C03651=1225.024,372.969,-76.050,-175.825,7.597,148.237
C03652=1225.028,372.721,-76.016,-175.826,7.594,148.237
C03653=1225.032,372.473,-75.983,-175.827,7.591,148.236
C03654=1225.036,372.225,-75.950,-175.829,7.588,148.236
C03655=1225.040,371.977,-75.917,-175.830,7.586,148.236
C03656=1225.044,371.730,-75.883,-175.831,7.583,148.235
C03657=1225.048,371.482,-75.850,-175.833,7.580,148.235
C03658=1225.052,371.234,-75.817,-175.834,7.577,148.235
C03659=1225.056,370.986,-75.784,-175.835,7.575,148.234
C03660=1225.061,370.739,-75.751,-175.837,7.572,148.234
C03661=1225.065,370.491,-75.718,-175.838,7.569,148.234
C03662=1225.069,370.243,-75.684,-175.839,7.566,148.233
C03663=1225.073,369.995,-75.651,-175.841,7.564,148.233
C03664=1225.077,369.748,-75.618,-175.842,7.561,148.233
C03665=1225.081,369.500,-75.585,-175.843,7.558,148.232
C03666=1225.085,369.252,-75.552,-175.844,7.555,148.232
C03667=1225.090,369.005,-75.519,-175.846,7.553,148.232
C03668=1225.094,368.756,-75.486,-175.847,7.550,148.231
C03669=1225.097,368.509,-75.454,-175.848,7.547,148.231
C03670=1225.101,368.261,-75.421,-175.850,7.544,148.231
C03671=1225.106,368.013,-75.387,-175.851,7.542,148.230
C03672=1225.110,367.766,-75.354,-175.852,7.539,148.230
C03673=1225.114,367.486,-75.317,-175.854,7.535,148.230
C03674=1225.120,367.207,-75.280,-175.856,7.533,148.229
C03675=1225.124,366.927,-75.243,-175.857,7.529,148.229
C03676=1225.129,366.647,-75.205,-175.859,7.527,148.229
C03677=1225.134,366.399,-75.173,-175.860,7.524,148.228
C03678=1225.137,366.152,-75.140,-175.861,7.521,148.228
C03679=1225.141,365.904,-75.107,-175.863,7.519,148.228
C03680=1225.145,365.656,-75.074,-175.864,7.516,148.227
C03681=1225.150,365.408,-75.041,-175.866,7.512,148.227
C03682=1225.154,365.160,-75.008,-175.868,7.510,148.227
C03683=1225.158,364.912,-74.975,-175.869,7.507,148.227
C03684=1225.161,364.665,-74.943,-175.870,7.504,148.226
C03685=1225.166,364.417,-74.910,-175.872,7.502,148.226
C03686=1225.170,364.169,-74.877,-175.873,7.499,148.226
C03687=1225.174,363.921,-74.844,-175.875,7.496,148.225
C03688=1225.178,363.673,-74.811,-175.876,7.494,148.225
C03689=1225.183,363.425,-74.778,-175.878,7.490,148.225
C03690=1225.186,363.178,-74.746,-175.880,7.488,148.225
C03691=1225.191,362.931,-74.713,-175.881,7.485,148.224
C03692=1225.195,362.682,-74.680,-175.883,7.482,148.224
C03693=1225.199,362.435,-74.647,-175.884,7.479,148.224
C03694=1225.203,362.186,-74.615,-175.885,7.477,148.223
C03695=1225.207,361.939,-74.582,-175.887,7.474,148.223
C03696=1225.211,361.691,-74.549,-175.889,7.471,148.223
C03697=1225.216,361.443,-74.517,-175.890,7.468,148.223
C03698=1225.219,361.195,-74.484,-175.892,7.465,148.222
C03699=1225.224,360.947,-74.452,-175.893,7.463,148.222
C03700=1225.228,360.700,-74.419,-175.895,7.460,148.222
C03701=1225.232,360.452,-74.386,-175.896,7.458,148.221
C03702=1225.236,360.204,-74.354,-175.898,7.454,148.221
C03703=1225.240,359.956,-74.321,-175.900,7.452,148.221
C03704=1225.245,359.708,-74.288,-175.901,7.449,148.221
C03705=1225.249,359.460,-74.255,-175.903,7.446,148.220
C03706=1225.253,359.212,-74.223,-175.904,7.444,148.220
C03707=1225.257,358.965,-74.190,-175.906,7.440,148.220
C03708=1225.262,358.717,-74.158,-175.908,7.438,148.220
C03709=1225.265,358.469,-74.125,-175.909,7.435,148.219
C03710=1225.270,358.221,-74.093,-175.910,7.432,148.219
C03711=1225.274,357.973,-74.060,-175.912,7.430,148.219
C03712=1225.277,357.725,-74.028,-175.914,7.426,148.219
C03713=1225.282,357.478,-73.995,-175.916,7.424,148.218
C03714=1225.287,357.230,-73.963,-175.917,7.421,148.218
C03715=1225.290,356.982,-73.931,-175.919,7.418,148.218
C03716=1225.295,356.734,-73.898,-175.920,7.416,148.218
C03717=1225.298,356.486,-73.866,-175.922,7.413,148.217
C03718=1225.302,356.238,-73.833,-175.924,7.410,148.217
C03719=1225.307,355.991,-73.801,-175.925,7.407,148.217
C03720=1225.311,355.743,-73.769,-175.927,7.405,148.217
C03721=1225.315,355.495,-73.736,-175.929,7.401,148.216
C03722=1225.320,355.247,-73.703,-175.931,7.399,148.216
C03723=1225.323,354.999,-73.671,-175.932,7.396,148.216
C03724=1225.328,354.752,-73.639,-175.933,7.393,148.216
C03725=1225.332,354.504,-73.607,-175.936,7.390,148.215
C03726=1225.336,354.255,-73.574,-175.937,7.388,148.215
C03727=1225.340,354.008,-73.542,-175.939,7.385,148.215
C03728=1225.344,353.759,-73.509,-175.941,7.382,148.215
C03729=1225.349,353.512,-73.477,-175.942,7.380,148.215
C03730=1225.353,353.264,-73.445,-175.944,7.377,148.214
C03731=1225.357,353.016,-73.412,-175.946,7.374,148.214
C03732=1225.361,352.768,-73.380,-175.947,7.371,148.214
C03733=1225.366,352.520,-73.348,-175.949,7.369,148.214
C03734=1225.369,352.273,-73.316,-175.951,7.365,148.213
C03735=1225.374,352.025,-73.283,-175.953,7.363,148.213
C03736=1225.377,351.777,-73.251,-175.954,7.360,148.213
C03737=1225.382,351.529,-73.219,-175.956,7.358,148.213
C03738=1225.386,351.281,-73.188,-175.958,7.354,148.213
C03739=1225.390,351.033,-73.154,-175.960,7.352,148.213
C03740=1225.395,350.786,-73.123,-175.961,7.349,148.212
C03741=1225.399,350.537,-73.091,-175.963,7.346,148.212
C03742=1225.403,350.289,-73.059,-175.965,7.343,148.212
C03743=1225.407,350.041,-73.026,-175.967,7.341,148.212
C03744=1225.411,349.794,-72.995,-175.968,7.338,148.212
C03745=1225.415,349.546,-72.963,-175.971,7.335,148.211
C03746=1225.419,349.298,-72.930,-175.972,7.333,148.211
C03747=1225.424,349.051,-72.898,-175.974,7.330,148.211
C03748=1225.428,348.802,-72.866,-175.975,7.327,148.211
C03749=1225.432,348.554,-72.834,-175.978,7.324,148.211
C03750=1225.437,348.307,-72.802,-175.979,7.322,148.210
C03751=1225.440,348.059,-72.770,-175.981,7.319,148.210
C03752=1225.444,347.810,-72.738,-175.983,7.316,148.210
C03753=1225.449,347.563,-72.706,-175.985,7.313,148.210
C03754=1225.453,347.315,-72.674,-175.986,7.311,148.210
C03755=1225.457,347.066,-72.642,-175.988,7.308,148.209
C03756=1225.462,346.819,-72.610,-175.990,7.305,148.209
C03757=1225.465,346.571,-72.579,-175.992,7.302,148.209
C03758=1225.470,346.323,-72.546,-175.993,7.300,148.209
C03759=1225.474,346.075,-72.515,-175.996,7.296,148.209
C03760=1225.478,345.827,-72.483,-175.998,7.294,148.209
C03761=1225.482,345.579,-72.450,-175.999,7.292,148.208
C03762=1225.487,345.332,-72.419,-176.001,7.289,148.208
C03763=1225.490,345.084,-72.387,-176.003,7.286,148.208
C03764=1225.495,344.835,-72.355,-176.005,7.283,148.208
C03765=1225.499,344.587,-72.324,-176.006,7.281,148.208
C03766=1225.503,344.339,-72.292,-176.009,7.277,148.207
C03767=1225.508,344.092,-72.260,-176.010,7.275,148.207
C03768=1225.512,343.844,-72.228,-176.012,7.273,148.207
C03769=1225.516,343.596,-72.196,-176.014,7.269,148.207
C03770=1225.521,343.348,-72.164,-176.016,7.267,148.207
C03771=1225.524,343.100,-72.132,-176.018,7.264,148.207
C03772=1225.529,342.852,-72.101,-176.019,7.262,148.207
C03773=1225.533,342.604,-72.070,-176.022,7.259,148.206
C03774=1225.537,342.355,-72.037,-176.024,7.256,148.206
C03775=1225.541,342.108,-72.006,-176.025,7.253,148.206
C03776=1225.545,341.860,-71.974,-176.027,7.250,148.206
C03777=1225.550,341.582,-71.939,-176.029,7.248,148.206
C03778=1225.555,341.305,-71.903,-176.032,7.244,148.206
C03779=1225.560,341.027,-71.868,-176.034,7.241,148.205
C03780=1225.564,340.749,-71.833,-176.036,7.238,148.205
C03781=1225.568,340.501,-71.801,-176.038,7.235,148.205
C03782=1225.573,340.253,-71.769,-176.040,7.233,148.205
C03783=1225.577,340.005,-71.738,-176.042,7.230,148.205
C03784=1225.581,339.757,-71.706,-176.044,7.227,148.205
C03785=1225.585,339.509,-71.674,-176.046,7.225,148.205
C03786=1225.590,339.261,-71.644,-176.048,7.222,148.204
C03787=1225.593,339.013,-71.612,-176.050,7.219,148.204
C03788=1225.598,338.766,-71.580,-176.051,7.216,148.204
C03789=1225.602,338.517,-71.548,-176.053,7.214,148.204
C03790=1225.607,338.270,-71.517,-176.055,7.211,148.204
C03791=1225.610,338.022,-71.485,-176.057,7.208,148.204
C03792=1225.615,337.774,-71.454,-176.059,7.206,148.204
C03793=1225.619,337.526,-71.423,-176.061,7.203,148.204
C03794=1225.623,337.278,-71.392,-176.063,7.200,148.203
C03795=1225.627,337.030,-71.360,-176.065,7.198,148.203
C03796=1225.631,336.782,-71.328,-176.067,7.195,148.203
C03797=1225.636,336.533,-71.297,-176.069,7.192,148.203
C03798=1225.640,336.286,-71.265,-176.071,7.190,148.203
C03799=1225.644,336.037,-71.234,-176.073,7.187,148.203
C03800=1225.649,335.790,-71.203,-176.075,7.184,148.203
C03801=1225.653,335.541,-71.172,-176.077,7.182,148.203
C03802=1225.657,335.294,-71.140,-176.079,7.178,148.202
C03803=1225.661,335.045,-71.109,-176.081,7.176,148.203
C03804=1225.665,334.798,-71.077,-176.083,7.174,148.202
C03805=1225.669,334.549,-71.046,-176.085,7.171,148.202
C03806=1225.674,334.302,-71.015,-176.087,7.168,148.202
C03807=1225.678,334.053,-70.984,-176.089,7.166,148.202
C03808=1225.682,333.806,-70.952,-176.091,7.162,148.202
C03809=1225.686,333.557,-70.921,-176.093,7.160,148.202
C03810=1225.691,333.310,-70.890,-176.096,7.157,148.202
C03811=1225.695,333.062,-70.859,-176.097,7.154,148.202
C03812=1225.699,332.814,-70.828,-176.099,7.152,148.202
C03813=1225.703,332.566,-70.796,-176.102,7.149,148.201
C03814=1225.707,332.318,-70.765,-176.104,7.147,148.201
C03815=1225.712,332.070,-70.734,-176.105,7.144,148.201
C03816=1225.716,331.822,-70.702,-176.108,7.141,148.201
C03817=1225.720,331.574,-70.672,-176.110,7.138,148.201
C03818=1225.725,331.326,-70.641,-176.112,7.136,148.201
C03819=1225.729,331.078,-70.609,-176.114,7.133,148.201
C03820=1225.733,330.830,-70.578,-176.116,7.131,148.201
C03821=1225.737,330.581,-70.547,-176.118,7.128,148.201
C03822=1225.741,330.333,-70.517,-176.120,7.125,148.201
C03823=1225.745,330.086,-70.486,-176.122,7.123,148.201
C03824=1225.749,329.837,-70.454,-176.124,7.120,148.201
C03825=1225.754,329.589,-70.424,-176.126,7.117,148.200
C03826=1225.759,329.341,-70.393,-176.128,7.115,148.200
C03827=1225.762,329.093,-70.361,-176.130,7.112,148.200
C03828=1225.767,328.845,-70.330,-176.133,7.109,148.200
C03829=1225.772,328.597,-70.300,-176.134,7.107,148.200
C03830=1225.775,328.349,-70.269,-176.136,7.104,148.200
C03831=1225.779,328.101,-70.238,-176.139,7.101,148.200
C03832=1225.783,327.853,-70.206,-176.141,7.099,148.200
C03833=1225.788,327.605,-70.176,-176.143,7.097,148.200
C03834=1225.792,327.357,-70.145,-176.145,7.093,148.200
C03835=1225.796,327.109,-70.114,-176.147,7.091,148.200
C03836=1225.800,326.861,-70.084,-176.149,7.088,148.200
C03837=1225.805,326.613,-70.053,-176.151,7.085,148.200
C03838=1225.809,326.364,-70.022,-176.153,7.083,148.200
C03839=1225.813,326.116,-69.991,-176.156,7.080,148.199
C03840=1225.818,325.869,-69.959,-176.158,7.078,148.199
C03841=1225.822,325.621,-69.929,-176.160,7.075,148.200
C03842=1225.826,325.373,-69.898,-176.162,7.072,148.199
C03843=1225.830,325.125,-69.867,-176.164,7.070,148.199
C03844=1225.835,324.877,-69.837,-176.166,7.067,148.199
C03845=1225.838,324.628,-69.806,-176.168,7.064,148.199
C03846=1225.843,324.380,-69.775,-176.170,7.062,148.199
C03847=1225.847,324.132,-69.745,-176.172,7.059,148.199
C03848=1225.851,323.884,-69.713,-176.175,7.056,148.199
C03849=1225.855,323.636,-69.683,-176.177,7.054,148.199
C03850=1225.860,323.388,-69.652,-176.179,7.052,148.199
C03851=1225.865,323.140,-69.622,-176.181,7.049,148.199
C03852=1225.868,322.892,-69.591,-176.183,7.046,148.199
C03853=1225.872,322.644,-69.560,-176.185,7.044,148.199
C03854=1225.877,322.395,-69.530,-176.187,7.041,148.199
C03855=1225.881,322.148,-69.500,-176.190,7.039,148.199
C03856=1225.885,321.899,-69.469,-176.192,7.036,148.199
C03857=1225.890,321.651,-69.438,-176.194,7.033,148.199
C03858=1225.894,321.403,-69.408,-176.196,7.031,148.199
C03859=1225.898,321.155,-69.377,-176.199,7.028,148.199
C03860=1225.902,320.907,-69.346,-176.201,7.025,148.199
C03861=1225.906,320.659,-69.316,-176.202,7.023,148.199
C03862=1225.911,320.411,-69.286,-176.205,7.020,148.199
C03863=1225.915,320.163,-69.256,-176.207,7.018,148.199
C03864=1225.920,319.915,-69.225,-176.209,7.015,148.199
C03865=1225.924,319.666,-69.194,-176.211,7.012,148.198
C03866=1225.928,319.419,-69.164,-176.213,7.010,148.198
C03867=1225.932,319.170,-69.134,-176.216,7.008,148.199
C03868=1225.936,318.922,-69.104,-176.218,7.005,148.199
C03869=1225.941,318.675,-69.073,-176.220,7.002,148.199
C03870=1225.944,318.426,-69.042,-176.222,7.000,148.198
C03871=1225.949,318.178,-69.012,-176.225,6.997,148.198
C03872=1225.954,317.930,-68.981,-176.227,6.995,148.198
C03873=1225.958,317.682,-68.951,-176.229,6.992,148.198
C03874=1225.963,317.433,-68.921,-176.231,6.989,148.198
C03875=1225.966,317.186,-68.891,-176.233,6.987,148.198
C03876=1225.970,316.937,-68.860,-176.235,6.985,148.198
C03877=1225.974,316.689,-68.830,-176.238,6.981,148.198
C03878=1225.979,316.441,-68.800,-176.240,6.979,148.198
C03879=1225.983,316.193,-68.770,-176.242,6.977,148.198
C03880=1225.988,315.945,-68.740,-176.245,6.974,148.198
C03881=1225.992,315.669,-68.706,-176.247,6.971,148.198
C03882=1225.997,315.393,-68.672,-176.249,6.968,148.198
C03883=1226.001,315.117,-68.639,-176.252,6.965,148.198
C03884=1226.007,314.842,-68.605,-176.254,6.962,148.198
C03885=1226.011,314.594,-68.575,-176.256,6.960,148.198
C03886=1226.015,314.346,-68.544,-176.259,6.958,148.198
C03887=1226.019,314.097,-68.515,-176.261,6.955,148.198
C03888=1226.024,313.849,-68.484,-176.263,6.953,148.198
C03889=1226.028,313.601,-68.454,-176.265,6.950,148.198
C03890=1226.032,313.353,-68.424,-176.268,6.947,148.198
C03891=1226.037,313.105,-68.394,-176.270,6.945,148.199
C03892=1226.040,312.857,-68.364,-176.272,6.943,148.198
C03893=1226.045,312.608,-68.334,-176.274,6.939,148.198
C03894=1226.049,312.361,-68.304,-176.277,6.937,148.198
C03895=1226.053,312.112,-68.274,-176.279,6.935,148.198
C03896=1226.058,311.864,-68.244,-176.281,6.932,148.198
C03897=1226.062,311.616,-68.214,-176.283,6.930,148.199
C03898=1226.067,311.368,-68.184,-176.286,6.928,148.199
C03899=1226.070,311.119,-68.154,-176.288,6.924,148.199
C03900=1226.075,310.871,-68.124,-176.290,6.922,148.199
C03901=1226.079,310.622,-68.094,-176.292,6.920,148.199
C03902=1226.083,310.375,-68.064,-176.295,6.917,148.199
C03903=1226.087,310.126,-68.034,-176.297,6.915,148.199
C03904=1226.092,309.879,-68.004,-176.299,6.913,148.199
C03905=1226.096,309.630,-67.974,-176.302,6.909,148.199
C03906=1226.100,309.382,-67.945,-176.304,6.907,148.199
C03907=1226.105,309.134,-67.915,-176.306,6.905,148.199
C03908=1226.109,308.886,-67.885,-176.309,6.902,148.199
C03909=1226.113,308.638,-67.855,-176.311,6.900,148.199
C03910=1226.118,308.389,-67.826,-176.313,6.898,148.199
C03911=1226.122,308.141,-67.795,-176.316,6.894,148.199
C03912=1226.126,307.893,-67.765,-176.318,6.892,148.199
C03913=1226.131,307.645,-67.736,-176.320,6.890,148.199
C03914=1226.135,307.396,-67.707,-176.323,6.887,148.199
C03915=1226.139,307.149,-67.676,-176.325,6.885,148.199
C03916=1226.144,306.900,-67.646,-176.327,6.883,148.199
C03917=1226.148,306.652,-67.617,-176.329,6.879,148.199
C03918=1226.152,306.404,-67.587,-176.331,6.877,148.199
C03919=1226.156,306.155,-67.558,-176.334,6.875,148.199
C03920=1226.161,305.907,-67.528,-176.336,6.872,148.199
C03921=1226.166,305.660,-67.498,-176.338,6.870,148.199
C03922=1226.170,305.412,-67.469,-176.340,6.868,148.199
C03923=1226.174,305.163,-67.439,-176.343,6.865,148.199
C03924=1226.178,304.915,-67.410,-176.345,6.862,148.199
C03925=1226.182,304.667,-67.380,-176.347,6.860,148.200
C03926=1226.187,304.418,-67.350,-176.350,6.857,148.200
C03927=1226.191,304.170,-67.321,-176.352,6.855,148.200
C03928=1226.196,303.922,-67.291,-176.354,6.853,148.200
C03929=1226.200,303.673,-67.262,-176.357,6.850,148.200
C03930=1226.204,303.425,-67.232,-176.359,6.847,148.200
C03931=1226.208,303.177,-67.203,-176.362,6.845,148.200
C03932=1226.212,302.929,-67.173,-176.364,6.843,148.200
C03933=1226.217,302.681,-67.143,-176.366,6.840,148.200
C03934=1226.222,302.433,-67.114,-176.368,6.838,148.200
C03935=1226.226,302.185,-67.084,-176.371,6.836,148.200
C03936=1226.230,301.937,-67.055,-176.373,6.833,148.200
C03937=1226.235,301.688,-67.026,-176.375,6.830,148.200
C03938=1226.239,301.439,-66.997,-176.377,6.828,148.200
C03939=1226.243,301.191,-66.967,-176.380,6.825,148.200
C03940=1226.247,300.943,-66.938,-176.383,6.823,148.201
C03941=1226.251,300.695,-66.908,-176.385,6.821,148.201
C03942=1226.256,300.447,-66.879,-176.387,6.818,148.201
C03943=1226.260,300.199,-66.850,-176.390,6.816,148.201
C03944=1226.264,299.951,-66.820,-176.392,6.814,148.201
C03945=1226.269,299.702,-66.791,-176.394,6.811,148.201
C03946=1226.273,299.454,-66.761,-176.396,6.808,148.201
C03947=1226.277,299.206,-66.732,-176.399,6.806,148.201
C03948=1226.281,298.957,-66.703,-176.401,6.804,148.201
C03949=1226.286,298.709,-66.674,-176.404,6.801,148.201
C03950=1226.290,298.461,-66.645,-176.406,6.799,148.201
C03951=1226.295,298.213,-66.615,-176.408,6.797,148.201
C03952=1226.299,297.965,-66.586,-176.411,6.794,148.201
C03953=1226.303,297.716,-66.557,-176.413,6.792,148.202
C03954=1226.308,297.468,-66.528,-176.415,6.790,148.202
C03955=1226.312,297.220,-66.498,-176.417,6.787,148.202
C03956=1226.316,296.972,-66.469,-176.420,6.784,148.202
C03957=1226.321,296.723,-66.440,-176.422,6.782,148.202
C03958=1226.324,296.475,-66.411,-176.424,6.780,148.202
C03959=1226.329,296.227,-66.382,-176.427,6.777,148.202
C03960=1226.333,295.979,-66.353,-176.430,6.775,148.202
C03961=1226.338,295.730,-66.324,-176.432,6.773,148.202
C03962=1226.342,295.482,-66.295,-176.434,6.770,148.202
C03963=1226.346,295.233,-66.265,-176.437,6.768,148.202
C03964=1226.351,294.985,-66.237,-176.439,6.765,148.203
C03965=1226.355,294.737,-66.207,-176.441,6.763,148.203
C03966=1226.359,294.489,-66.178,-176.444,6.760,148.203
C03967=1226.363,294.240,-66.150,-176.446,6.758,148.203
C03968=1226.368,293.993,-66.121,-176.449,6.756,148.203
C03969=1226.373,293.744,-66.092,-176.451,6.754,148.203
C03970=1226.377,293.495,-66.062,-176.453,6.751,148.203
C03971=1226.381,293.247,-66.033,-176.455,6.749,148.203
C03972=1226.385,292.999,-66.005,-176.458,6.747,148.203
C03973=1226.389,292.751,-65.976,-176.460,6.744,148.203
C03974=1226.394,292.502,-65.947,-176.463,6.741,148.203
C03975=1226.399,292.255,-65.918,-176.465,6.739,148.203
C03976=1226.403,292.006,-65.890,-176.468,6.737,148.204
C03977=1226.407,291.758,-65.860,-176.470,6.734,148.204
C03978=1226.411,291.509,-65.832,-176.472,6.732,148.204
C03979=1226.416,291.261,-65.803,-176.475,6.730,148.204
C03980=1226.420,291.012,-65.774,-176.477,6.728,148.204
C03981=1226.424,290.764,-65.745,-176.480,6.725,148.204
C03982=1226.429,290.516,-65.717,-176.482,6.723,148.204
C03983=1226.433,290.268,-65.687,-176.484,6.721,148.205
C03984=1226.437,290.019,-65.659,-176.486,6.719,148.205
C03985=1226.442,289.745,-65.627,-176.489,6.715,148.205
C03986=1226.447,289.472,-65.595,-176.492,6.713,148.205
C03987=1226.452,289.198,-65.564,-176.494,6.711,148.205
C03988=1226.456,288.923,-65.532,-176.498,6.708,148.205
C03989=1226.461,288.674,-65.503,-176.500,6.706,148.205
C03990=1226.466,288.427,-65.474,-176.502,6.703,148.205
C03991=1226.469,288.178,-65.446,-176.504,6.701,148.206
C03992=1226.474,287.929,-65.417,-176.507,6.698,148.206
C03993=1226.479,287.682,-65.388,-176.509,6.696,148.206
C03994=1226.482,287.433,-65.360,-176.512,6.694,148.206
C03995=1226.487,287.184,-65.331,-176.514,6.692,148.206
C03996=1226.491,286.937,-65.303,-176.516,6.689,148.206
C03997=1226.495,286.688,-65.274,-176.519,6.687,148.206
C03998=1226.501,286.440,-65.246,-176.521,6.685,148.206
C03999=1226.504,286.191,-65.218,-176.523,6.683,148.206
C04000=1226.508,285.943,-65.188,-176.526,6.680,148.207
C04001=1226.513,285.695,-65.160,-176.529,6.678,148.207
C04002=1226.517,285.446,-65.132,-176.531,6.676,148.207
C04003=1226.522,285.198,-65.103,-176.533,6.674,148.207
C04004=1226.526,284.950,-65.074,-176.536,6.671,148.207
C04005=1226.531,284.702,-65.046,-176.539,6.669,148.207
C04006=1226.535,284.453,-65.018,-176.541,6.666,148.207
C04007=1226.539,284.205,-64.989,-176.543,6.664,148.208
C04008=1226.544,283.957,-64.961,-176.546,6.662,148.208
C04009=1226.548,283.708,-64.933,-176.548,6.659,148.208
C04010=1226.552,283.460,-64.905,-176.551,6.657,148.208
C04011=1226.557,283.212,-64.875,-176.553,6.655,148.208
C04012=1226.561,282.964,-64.848,-176.555,6.653,148.208
C04013=1226.565,282.715,-64.819,-176.558,6.650,148.208
C04014=1226.570,282.467,-64.791,-176.560,6.648,148.209
C04015=1226.574,282.218,-64.762,-176.563,6.646,148.209
C04016=1226.578,281.970,-64.734,-176.565,6.644,148.209
C04017=1226.583,281.721,-64.706,-176.567,6.642,148.209
C04018=1226.587,281.473,-64.678,-176.570,6.639,148.209
C04019=1226.592,281.225,-64.649,-176.572,6.637,148.209
C04020=1226.596,280.976,-64.621,-176.575,6.635,148.210
C04021=1226.601,280.728,-64.593,-176.577,6.633,148.210
C04022=1226.605,280.479,-64.565,-176.580,6.630,148.210
C04023=1226.609,280.231,-64.537,-176.582,6.628,148.210
C04024=1226.613,279.983,-64.508,-176.584,6.626,148.210
C04025=1226.618,279.735,-64.480,-176.587,6.624,148.210
C04026=1226.622,279.486,-64.452,-176.589,6.621,148.210
C04027=1226.627,279.238,-64.424,-176.592,6.619,148.211
C04028=1226.630,278.989,-64.396,-176.594,6.616,148.211
C04029=1226.635,278.741,-64.367,-176.597,6.615,148.211
C04030=1226.640,278.493,-64.340,-176.599,6.612,148.211
C04031=1226.644,278.244,-64.311,-176.602,6.610,148.211
C04032=1226.649,277.996,-64.284,-176.604,6.607,148.211
C04033=1226.653,277.747,-64.256,-176.606,6.605,148.211
C04034=1226.658,277.499,-64.227,-176.609,6.603,148.212
C04035=1226.661,277.251,-64.199,-176.611,6.601,148.212
C04036=1226.666,277.003,-64.171,-176.614,6.599,148.212
C04037=1226.670,276.754,-64.143,-176.616,6.596,148.212
C04038=1226.675,276.505,-64.116,-176.619,6.594,148.212
C04039=1226.679,276.257,-64.087,-176.621,6.592,148.212
C04040=1226.683,276.009,-64.060,-176.624,6.590,148.213
C04041=1226.688,275.761,-64.031,-176.626,6.588,148.213
C04042=1226.692,275.512,-64.003,-176.628,6.586,148.213
C04043=1226.697,275.264,-63.976,-176.631,6.583,148.213
C04044=1226.701,275.015,-63.947,-176.634,6.581,148.213
C04045=1226.705,274.767,-63.920,-176.636,6.579,148.214
C04046=1226.710,274.519,-63.892,-176.638,6.577,148.214
C04047=1226.714,274.270,-63.864,-176.640,6.575,148.214
C04048=1226.719,274.022,-63.836,-176.643,6.573,148.214
C04049=1226.723,273.773,-63.808,-176.646,6.570,148.214
C04050=1226.727,273.524,-63.781,-176.648,6.568,148.214
C04051=1226.732,273.277,-63.753,-176.650,6.566,148.215
C04052=1226.735,273.028,-63.725,-176.653,6.564,148.215
C04053=1226.741,272.779,-63.697,-176.655,6.562,148.215
C04054=1226.745,272.531,-63.669,-176.658,6.560,148.215
C04055=1226.749,272.283,-63.641,-176.660,6.557,148.215
C04056=1226.754,272.034,-63.614,-176.663,6.555,148.216
C04057=1226.758,271.786,-63.586,-176.665,6.553,148.216
C04058=1226.763,271.537,-63.558,-176.668,6.551,148.216
C04059=1226.767,271.289,-63.531,-176.670,6.549,148.216
C04060=1226.772,271.040,-63.504,-176.672,6.547,148.216
C04061=1226.775,270.792,-63.475,-176.676,6.544,148.217
C04062=1226.780,270.544,-63.448,-176.678,6.542,148.217
C04063=1226.784,270.296,-63.421,-176.680,6.540,148.217
C04064=1226.788,270.047,-63.392,-176.682,6.538,148.217
C04065=1226.793,269.798,-63.365,-176.685,6.536,148.217
C04066=1226.798,269.550,-63.337,-176.687,6.534,148.217
C04067=1226.802,269.301,-63.310,-176.690,6.532,148.218
C04068=1226.806,269.053,-63.282,-176.692,6.529,148.218
C04069=1226.811,268.805,-63.255,-176.695,6.527,148.218
C04070=1226.816,268.556,-63.228,-176.698,6.525,148.218
C04071=1226.819,268.308,-63.200,-176.700,6.523,148.218
C04072=1226.824,268.059,-63.172,-176.702,6.521,148.219
C04073=1226.828,267.811,-63.145,-176.704,6.518,148.219
C04074=1226.832,267.562,-63.117,-176.707,6.517,148.219
C04075=1226.837,267.314,-63.090,-176.710,6.514,148.219
C04076=1226.841,267.066,-63.062,-176.712,6.512,148.219
C04077=1226.846,266.817,-63.035,-176.715,6.510,148.220
C04078=1226.850,266.569,-63.007,-176.717,6.508,148.220
C04079=1226.855,266.320,-62.980,-176.720,6.506,148.220
C04080=1226.859,266.072,-62.953,-176.722,6.503,148.220
C04081=1226.864,265.824,-62.925,-176.724,6.502,148.220
C04082=1226.868,265.575,-62.898,-176.727,6.500,148.221
C04083=1226.872,265.326,-62.871,-176.730,6.497,148.221
C04084=1226.877,265.078,-62.843,-176.732,6.495,148.221
C04085=1226.881,264.830,-62.816,-176.734,6.493,148.221
C04086=1226.886,264.581,-62.789,-176.737,6.491,148.221
C04087=1226.890,264.332,-62.762,-176.740,6.489,148.222
C04088=1226.894,264.084,-62.734,-176.742,6.487,148.222
C04089=1226.900,263.811,-62.704,-176.745,6.484,148.222
C04090=1226.904,263.539,-62.674,-176.748,6.482,148.222
C04091=1226.909,263.266,-62.645,-176.750,6.480,148.223
C04092=1226.914,262.994,-62.614,-176.753,6.477,148.223
C04093=1226.919,262.745,-62.587,-176.755,6.475,148.223
C04094=1226.923,262.496,-62.560,-176.758,6.473,148.223
C04095=1226.928,262.247,-62.533,-176.760,6.471,148.223
C04096=1226.931,262.000,-62.506,-176.763,6.469,148.224
C04097=1226.936,261.751,-62.479,-176.765,6.467,148.224
C04098=1226.941,261.503,-62.452,-176.767,6.465,148.224
C04099=1226.945,261.254,-62.425,-176.770,6.463,148.224
C04100=1226.949,261.005,-62.397,-176.773,6.460,148.224
C04101=1226.954,260.757,-62.370,-176.775,6.458,148.225
C04102=1226.959,260.508,-62.343,-176.778,6.456,148.225
C04103=1226.962,260.260,-62.316,-176.780,6.454,148.225
C04104=1226.967,260.012,-62.289,-176.783,6.452,148.225
C04105=1226.972,259.763,-62.262,-176.785,6.450,148.226
C04106=1226.976,259.515,-62.235,-176.787,6.448,148.226
C04107=1226.980,259.266,-62.207,-176.790,6.446,148.226
C04108=1226.984,259.018,-62.181,-176.793,6.444,148.226
C04109=1226.989,258.769,-62.154,-176.795,6.442,148.226
C04110=1226.993,258.521,-62.127,-176.797,6.440,148.227
C04111=1226.998,258.272,-62.100,-176.800,6.438,148.227
C04112=1227.002,258.024,-62.073,-176.803,6.435,148.227
C04113=1227.007,257.776,-62.046,-176.805,6.433,148.227
C04114=1227.012,257.527,-62.020,-176.808,6.432,148.228
C04115=1227.016,257.278,-61.993,-176.810,6.429,148.228
C04116=1227.020,257.030,-61.966,-176.813,6.428,148.228
C04117=1227.024,256.781,-61.939,-176.815,6.426,148.228
C04118=1227.029,256.532,-61.912,-176.818,6.424,148.229
C04119=1227.034,256.284,-61.885,-176.820,6.422,148.229
C04120=1227.037,256.035,-61.858,-176.823,6.420,148.229
C04121=1227.042,255.787,-61.831,-176.825,6.418,148.229
C04122=1227.047,255.538,-61.804,-176.827,6.416,148.229
C04123=1227.051,255.290,-61.777,-176.830,6.414,148.230
C04124=1227.056,255.041,-61.751,-176.832,6.412,148.230
C04125=1227.060,254.793,-61.724,-176.835,6.410,148.230
C04126=1227.064,254.544,-61.698,-176.837,6.408,148.230
C04127=1227.069,254.296,-61.671,-176.840,6.406,148.231
C04128=1227.074,254.048,-61.644,-176.843,6.403,148.231
C04129=1227.078,253.799,-61.618,-176.845,6.401,148.231
C04130=1227.082,253.550,-61.591,-176.848,6.399,148.231
C04131=1227.087,253.302,-61.564,-176.850,6.397,148.232
C04132=1227.091,253.054,-61.537,-176.852,6.395,148.232
C04133=1227.096,252.804,-61.511,-176.855,6.393,148.232
C04134=1227.100,252.556,-61.484,-176.858,6.391,148.232
C04135=1227.105,252.308,-61.457,-176.860,6.389,148.233
C04136=1227.109,252.059,-61.430,-176.862,6.387,148.233
C04137=1227.113,251.810,-61.404,-176.865,6.385,148.233
C04138=1227.118,251.562,-61.377,-176.868,6.383,148.233
C04139=1227.122,251.314,-61.351,-176.870,6.381,148.234
C04140=1227.127,251.065,-61.325,-176.872,6.379,148.234
C04141=1227.131,250.816,-61.298,-176.875,6.377,148.234
C04142=1227.136,250.568,-61.271,-176.878,6.375,148.234
C04143=1227.140,250.319,-61.245,-176.880,6.373,148.234
C04144=1227.144,250.071,-61.218,-176.882,6.371,148.235
C04145=1227.149,249.822,-61.192,-176.885,6.370,148.235
C04146=1227.153,249.573,-61.165,-176.888,6.368,148.235
C04147=1227.158,249.325,-61.138,-176.890,6.365,148.236
C04148=1227.162,249.076,-61.113,-176.892,6.364,148.236
C04149=1227.167,248.828,-61.086,-176.895,6.362,148.236
C04150=1227.171,248.579,-61.060,-176.898,6.360,148.236
C04151=1227.176,248.331,-61.034,-176.900,6.358,148.237
C04152=1227.181,248.082,-61.007,-176.902,6.356,148.237
C04153=1227.184,247.834,-60.981,-176.905,6.354,148.237
C04154=1227.189,247.585,-60.955,-176.907,6.352,148.237
C04155=1227.193,247.337,-60.928,-176.910,6.350,148.238
C04156=1227.198,247.088,-60.902,-176.912,6.348,148.238
C04157=1227.202,246.839,-60.875,-176.915,6.346,148.238
C04158=1227.207,246.590,-60.849,-176.917,6.344,148.238
C04159=1227.211,246.342,-60.822,-176.920,6.342,148.239
C04160=1227.215,246.093,-60.797,-176.922,6.340,148.239
C04161=1227.221,245.845,-60.770,-176.925,6.338,148.239
C04162=1227.225,245.597,-60.744,-176.927,6.336,148.239
C04163=1227.229,245.348,-60.717,-176.930,6.334,148.240
C04164=1227.234,245.099,-60.691,-176.933,6.333,148.240
C04165=1227.238,244.851,-60.666,-176.935,6.330,148.240
C04166=1227.243,244.602,-60.639,-176.937,6.328,148.241
C04167=1227.247,244.353,-60.613,-176.940,6.327,148.241
C04168=1227.251,244.104,-60.587,-176.943,6.325,148.241
C04169=1227.256,243.857,-60.560,-176.945,6.323,148.241
C04170=1227.261,243.608,-60.535,-176.947,6.321,148.242
C04171=1227.265,243.359,-60.509,-176.950,6.319,148.242
C04172=1227.269,243.111,-60.482,-176.953,6.317,148.242
C04173=1227.274,242.862,-60.456,-176.955,6.315,148.242
C04174=1227.278,242.613,-60.430,-176.958,6.313,148.243
C04175=1227.283,242.365,-60.404,-176.960,6.311,148.243
C04176=1227.287,242.116,-60.378,-176.963,6.309,148.243
C04177=1227.292,241.868,-60.352,-176.965,6.307,148.244
C04178=1227.297,241.618,-60.326,-176.968,6.305,148.244
C04179=1227.300,241.370,-60.299,-176.970,6.303,148.244
C04180=1227.305,241.122,-60.274,-176.973,6.301,148.244
C04181=1227.309,240.873,-60.248,-176.975,6.299,148.245
C04182=1227.314,240.624,-60.222,-176.978,6.297,148.245
C04183=1227.319,240.375,-60.196,-176.980,6.296,148.245
C04184=1227.323,240.127,-60.170,-176.983,6.294,148.245
C04185=1227.327,239.879,-60.144,-176.986,6.292,148.246
C04186=1227.332,239.630,-60.118,-176.988,6.290,148.246
C04187=1227.337,239.381,-60.092,-176.990,6.288,148.246
C04188=1227.341,239.132,-60.066,-176.993,6.286,148.247
C04189=1227.346,238.884,-60.041,-176.996,6.284,148.247
C04190=1227.350,238.636,-60.015,-176.998,6.282,148.247
C04191=1227.355,238.387,-59.988,-177.001,6.280,148.247
C04192=1227.359,238.138,-59.963,-177.003,6.278,148.248
C04193=1227.364,237.867,-59.935,-177.006,6.276,148.248
C04194=1227.369,237.595,-59.907,-177.009,6.275,148.248
C04195=1227.374,237.325,-59.878,-177.011,6.273,148.249
C04196=1227.378,237.053,-59.850,-177.014,6.270,148.249
C04197=1227.383,236.804,-59.825,-177.017,6.268,148.249
C04198=1227.387,236.556,-59.799,-177.019,6.266,148.249
C04199=1227.392,236.307,-59.773,-177.022,6.264,148.250
C04200=1227.397,236.058,-59.747,-177.024,6.263,148.250
C04201=1227.401,235.810,-59.722,-177.027,6.261,148.250
C04202=1227.406,235.561,-59.696,-177.029,6.259,148.251
C04203=1227.410,235.312,-59.670,-177.032,6.257,148.251
C04204=1227.415,235.064,-59.645,-177.034,6.256,148.251
C04205=1227.419,234.815,-59.619,-177.037,6.253,148.251
C04206=1227.423,234.566,-59.593,-177.039,6.251,148.252
C04207=1227.427,234.318,-59.568,-177.042,6.250,148.252
C04208=1227.432,234.069,-59.542,-177.044,6.248,148.252
C04209=1227.436,233.821,-59.516,-177.047,6.246,148.253
C04210=1227.441,233.572,-59.491,-177.050,6.244,148.253
C04211=1227.446,233.323,-59.466,-177.052,6.242,148.253
C04212=1227.450,233.074,-59.440,-177.055,6.240,148.254
C04213=1227.455,232.826,-59.415,-177.057,6.238,148.254
C04214=1227.460,232.577,-59.389,-177.060,6.236,148.254
C04215=1227.464,232.328,-59.363,-177.062,6.234,148.254
C04216=1227.469,232.080,-59.337,-177.064,6.233,148.255
C04217=1227.473,231.831,-59.312,-177.067,6.231,148.255
C04218=1227.478,231.582,-59.287,-177.070,6.230,148.255
C04219=1227.482,231.334,-59.261,-177.072,6.228,148.256
C04220=1227.486,231.085,-59.236,-177.075,6.226,148.256
C04221=1227.490,230.837,-59.210,-177.077,6.224,148.256
C04222=1227.495,230.588,-59.186,-177.080,6.222,148.257
C04223=1227.500,230.339,-59.160,-177.082,6.220,148.257
C04224=1227.504,230.091,-59.135,-177.085,6.218,148.257
C04225=1227.509,229.842,-59.109,-177.087,6.216,148.257
C04226=1227.513,229.593,-59.084,-177.090,6.214,148.258
C04227=1227.518,229.345,-59.058,-177.093,6.212,148.258
C04228=1227.522,229.096,-59.033,-177.095,6.211,148.258
C04229=1227.527,228.848,-59.007,-177.097,6.209,148.259
C04230=1227.532,228.598,-58.982,-177.100,6.208,148.259
C04231=1227.536,228.350,-58.957,-177.103,6.206,148.259
C04232=1227.541,228.101,-58.931,-177.105,6.204,148.260
C04233=1227.545,227.852,-58.906,-177.108,6.202,148.260
C04234=1227.549,227.604,-58.881,-177.110,6.200,148.260
C04235=1227.554,227.355,-58.856,-177.113,6.198,148.260
C04236=1227.559,227.107,-58.831,-177.115,6.196,148.261
C04237=1227.563,226.858,-58.805,-177.118,6.194,148.261
C04238=1227.568,226.609,-58.780,-177.120,6.192,148.261
C04239=1227.572,226.360,-58.755,-177.123,6.190,148.262
C04240=1227.577,226.112,-58.731,-177.125,6.189,148.262
C04241=1227.581,225.863,-58.705,-177.128,6.188,148.262
C04242=1227.586,225.615,-58.679,-177.130,6.186,148.263
C04243=1227.590,225.366,-58.654,-177.133,6.184,148.263
C04244=1227.595,225.117,-58.629,-177.136,6.182,148.263
C04245=1227.599,224.868,-58.604,-177.138,6.180,148.264
C04246=1227.604,224.620,-58.579,-177.141,6.178,148.264
C04247=1227.608,224.371,-58.554,-177.144,6.176,148.264
C04248=1227.613,224.123,-58.529,-177.146,6.174,148.265
C04249=1227.617,223.873,-58.504,-177.148,6.173,148.265
C04250=1227.622,223.625,-58.479,-177.151,6.172,148.265
C04251=1227.626,223.376,-58.454,-177.153,6.170,148.266
C04252=1227.631,223.127,-58.429,-177.156,6.168,148.266
C04253=1227.635,222.879,-58.403,-177.159,6.166,148.266
C04254=1227.640,222.630,-58.379,-177.161,6.164,148.267
C04255=1227.644,222.381,-58.354,-177.164,6.162,148.267
C04256=1227.649,222.133,-58.329,-177.167,6.160,148.267
C04257=1227.654,221.883,-58.304,-177.169,6.159,148.268
C04258=1227.658,221.635,-58.279,-177.171,6.158,148.268
C04259=1227.662,221.386,-58.254,-177.173,6.155,148.268
C04260=1227.667,221.138,-58.229,-177.176,6.153,148.269
C04261=1227.672,220.889,-58.205,-177.179,6.152,148.269
C04262=1227.676,220.640,-58.180,-177.181,6.150,148.269
C04263=1227.681,220.392,-58.154,-177.184,6.148,148.269
C04264=1227.685,220.143,-58.130,-177.187,6.146,148.270
C04265=1227.690,219.894,-58.105,-177.189,6.144,148.270
C04266=1227.694,219.645,-58.080,-177.191,6.143,148.271
C04267=1227.698,219.397,-58.055,-177.194,6.141,148.271
C04268=1227.704,219.148,-58.031,-177.197,6.139,148.271
C04269=1227.707,218.899,-58.006,-177.199,6.138,148.271
C04270=1227.712,218.651,-57.981,-177.202,6.136,148.272
C04271=1227.717,218.401,-57.956,-177.204,6.134,148.272
C04272=1227.721,218.153,-57.932,-177.207,6.132,148.272
C04273=1227.726,217.904,-57.907,-177.210,6.130,148.273
C04274=1227.730,217.655,-57.883,-177.212,6.129,148.273
C04275=1227.735,217.407,-57.857,-177.214,6.127,148.273
C04276=1227.739,217.158,-57.832,-177.217,6.125,148.274
C04277=1227.744,216.909,-57.808,-177.220,6.123,148.274
C04278=1227.749,216.661,-57.783,-177.223,6.122,148.275
C04279=1227.753,216.411,-57.759,-177.225,6.120,148.275
C04280=1227.758,216.163,-57.734,-177.228,6.118,148.275
C04281=1227.762,215.915,-57.710,-177.230,6.117,148.276
C04282=1227.766,215.665,-57.685,-177.233,6.115,148.276
C04283=1227.771,215.417,-57.660,-177.235,6.113,148.276
C04284=1227.776,215.168,-57.636,-177.238,6.112,148.277
C04285=1227.780,214.919,-57.611,-177.241,6.110,148.277
C04286=1227.785,214.671,-57.587,-177.243,6.108,148.277
C04287=1227.789,214.422,-57.563,-177.246,6.106,148.278
C04288=1227.794,214.173,-57.538,-177.248,6.105,148.278
C04289=1227.798,213.924,-57.513,-177.251,6.103,148.278
C04290=1227.803,213.676,-57.489,-177.253,6.101,148.279
C04291=1227.807,213.426,-57.464,-177.256,6.099,148.279
C04292=1227.812,213.178,-57.440,-177.258,6.098,148.279
C04293=1227.817,212.929,-57.416,-177.261,6.096,148.280
C04294=1227.821,212.680,-57.391,-177.264,6.094,148.280
C04295=1227.826,212.431,-57.367,-177.266,6.093,148.280
C04296=1227.831,212.183,-57.342,-177.268,6.091,148.281
C04297=1227.835,211.913,-57.316,-177.271,6.089,148.281
C04298=1227.840,211.642,-57.289,-177.274,6.088,148.282
C04299=1227.845,211.372,-57.262,-177.277,6.086,148.282
C04300=1227.850,211.101,-57.236,-177.279,6.084,148.282
C04301=1227.855,210.853,-57.212,-177.282,6.082,148.283
C04302=1227.860,210.604,-57.187,-177.285,6.080,148.283
C04303=1227.864,210.355,-57.163,-177.287,6.078,148.283
C04304=1227.868,210.106,-57.139,-177.290,6.076,148.284
C04305=1227.873,209.858,-57.114,-177.293,6.074,148.284
C04306=1227.878,209.609,-57.090,-177.295,6.073,148.284
C04307=1227.882,209.360,-57.066,-177.298,6.072,148.285
C04308=1227.887,209.111,-57.042,-177.300,6.070,148.285
C04309=1227.891,208.862,-57.017,-177.303,6.068,148.286
C04310=1227.896,208.614,-56.993,-177.306,6.066,148.286
C04311=1227.900,208.365,-56.968,-177.308,6.065,148.286
C04312=1227.905,208.116,-56.945,-177.310,6.063,148.287
C04313=1227.909,207.867,-56.921,-177.313,6.062,148.287
C04314=1227.914,207.618,-56.896,-177.316,6.060,148.287
C04315=1227.919,207.370,-56.872,-177.318,6.058,148.288
C04316=1227.923,207.121,-56.848,-177.321,6.056,148.288
C04317=1227.928,206.872,-56.824,-177.323,6.055,148.288
C04318=1227.932,206.623,-56.800,-177.326,6.053,148.289
C04319=1227.937,206.375,-56.776,-177.328,6.051,148.289
C04320=1227.941,206.126,-56.752,-177.331,6.050,148.290
C04321=1227.947,205.877,-56.728,-177.333,6.049,148.290
C04322=1227.950,205.628,-56.703,-177.336,6.047,148.290
C04323=1227.955,205.379,-56.679,-177.339,6.045,148.291
C04324=1227.959,205.130,-56.656,-177.341,6.043,148.291
C04325=1227.965,204.882,-56.631,-177.344,6.041,148.291
C04326=1227.969,204.633,-56.607,-177.346,6.040,148.292
C04327=1227.974,204.384,-56.584,-177.349,6.038,148.292
C04328=1227.977,204.135,-56.559,-177.351,6.037,148.292
C04329=1227.982,203.886,-56.536,-177.354,6.035,148.293
C04330=1227.987,203.637,-56.511,-177.357,6.033,148.293
C04331=1227.992,203.389,-56.487,-177.359,6.032,148.294
C04332=1227.996,203.140,-56.464,-177.362,6.030,148.294
C04333=1228.001,202.891,-56.440,-177.364,6.029,148.294
C04334=1228.006,202.642,-56.416,-177.367,6.027,148.295
C04335=1228.010,202.394,-56.392,-177.369,6.026,148.295
C04336=1228.015,202.144,-56.368,-177.372,6.024,148.295
C04337=1228.019,201.896,-56.344,-177.374,6.022,148.296
C04338=1228.024,201.647,-56.320,-177.377,6.020,148.296
C04339=1228.028,201.398,-56.296,-177.379,6.019,148.296
C04340=1228.033,201.150,-56.272,-177.382,6.018,148.297
C04341=1228.037,200.901,-56.249,-177.385,6.016,148.297
C04342=1228.042,200.652,-56.225,-177.388,6.014,148.298
C04343=1228.046,200.403,-56.202,-177.390,6.012,148.298
C04344=1228.051,200.154,-56.178,-177.392,6.011,148.298
C04345=1228.056,199.905,-56.154,-177.395,6.009,148.299
C04346=1228.061,199.656,-56.130,-177.398,6.007,148.299
C04347=1228.065,199.408,-56.106,-177.400,6.005,148.299
C04348=1228.069,199.158,-56.082,-177.403,6.005,148.300
C04349=1228.074,198.910,-56.058,-177.405,6.003,148.300
C04350=1228.079,198.661,-56.035,-177.408,6.001,148.301
C04351=1228.083,198.412,-56.012,-177.411,5.999,148.301
C04352=1228.088,198.163,-55.987,-177.413,5.998,148.301
C04353=1228.092,197.914,-55.964,-177.415,5.996,148.302
C04354=1228.097,197.665,-55.941,-177.418,5.994,148.302
C04355=1228.101,197.417,-55.917,-177.421,5.994,148.303
C04356=1228.106,197.168,-55.893,-177.423,5.992,148.303
C04357=1228.111,196.919,-55.870,-177.426,5.990,148.303
C04358=1228.115,196.670,-55.846,-177.428,5.988,148.304
C04359=1228.120,196.421,-55.823,-177.431,5.987,148.304
C04360=1228.125,196.172,-55.799,-177.433,5.985,148.304
C04361=1228.129,195.924,-55.775,-177.436,5.983,148.305
C04362=1228.134,195.675,-55.752,-177.439,5.982,148.305
C04363=1228.138,195.426,-55.728,-177.441,5.981,148.306
C04364=1228.143,195.177,-55.705,-177.444,5.979,148.306
C04365=1228.148,194.928,-55.681,-177.446,5.977,148.306
C04366=1228.152,194.679,-55.658,-177.448,5.976,148.307
C04367=1228.157,194.430,-55.634,-177.451,5.974,148.307
C04368=1228.162,194.181,-55.611,-177.454,5.973,148.307
C04369=1228.166,193.933,-55.587,-177.457,5.971,148.308
C04370=1228.170,193.684,-55.564,-177.459,5.970,148.308
C04371=1228.175,193.435,-55.541,-177.462,5.968,148.309
C04372=1228.179,193.186,-55.517,-177.464,5.966,148.309
C04373=1228.185,192.938,-55.494,-177.466,5.965,148.309
C04374=1228.189,192.689,-55.471,-177.469,5.963,148.310
C04375=1228.194,192.440,-55.447,-177.472,5.962,148.310
C04376=1228.198,192.191,-55.424,-177.475,5.960,148.311
C04377=1228.203,191.942,-55.400,-177.477,5.959,148.311
C04378=1228.207,191.694,-55.377,-177.479,5.957,148.311
C04379=1228.212,191.445,-55.354,-177.482,5.955,148.312
C04380=1228.217,191.196,-55.331,-177.485,5.955,148.312
C04381=1228.221,190.947,-55.307,-177.487,5.953,148.313
C04382=1228.226,190.697,-55.284,-177.490,5.951,148.313
C04383=1228.231,190.448,-55.261,-177.492,5.950,148.313
C04384=1228.235,190.200,-55.238,-177.495,5.948,148.314
C04385=1228.240,189.951,-55.215,-177.497,5.946,148.314
C04386=1228.245,189.702,-55.191,-177.500,5.945,148.315
C04387=1228.249,189.453,-55.168,-177.503,5.944,148.315
C04388=1228.254,189.204,-55.145,-177.505,5.942,148.315
C04389=1228.258,188.956,-55.122,-177.508,5.940,148.316
C04390=1228.263,188.707,-55.099,-177.510,5.939,148.316
C04391=1228.267,188.458,-55.075,-177.513,5.938,148.317
C04392=1228.272,188.208,-55.052,-177.516,5.936,148.317
C04393=1228.277,187.960,-55.030,-177.518,5.935,148.318
C04394=1228.281,187.711,-55.006,-177.520,5.933,148.318
C04395=1228.286,187.462,-54.983,-177.523,5.931,148.318
C04396=1228.291,187.213,-54.959,-177.526,5.930,148.319
C04397=1228.295,186.965,-54.937,-177.528,5.928,148.319
C04398=1228.299,186.716,-54.913,-177.531,5.927,148.319
C04399=1228.304,186.467,-54.890,-177.533,5.926,148.320
C04400=1228.309,186.218,-54.867,-177.536,5.924,148.320
C04401=1228.314,185.949,-54.843,-177.539,5.922,148.321
C04402=1228.319,185.678,-54.817,-177.541,5.920,148.321
C04403=1228.324,185.409,-54.792,-177.545,5.919,148.322
C04404=1228.329,185.139,-54.768,-177.547,5.917,148.322
C04405=1228.334,184.891,-54.745,-177.549,5.916,148.322
C04406=1228.339,184.642,-54.721,-177.552,5.914,148.323
C04407=1228.343,184.393,-54.699,-177.555,5.914,148.323
C04408=1228.348,184.143,-54.676,-177.557,5.912,148.324
C04409=1228.352,183.895,-54.653,-177.560,5.910,148.324
C04410=1228.357,183.646,-54.630,-177.562,5.909,148.325
C04411=1228.362,183.397,-54.607,-177.565,5.907,148.325
C04412=1228.366,183.148,-54.585,-177.568,5.905,148.325
C04413=1228.370,182.899,-54.561,-177.570,5.904,148.326
C04414=1228.374,182.650,-54.539,-177.572,5.903,148.326
C04415=1228.380,182.402,-54.516,-177.575,5.901,148.327
C04416=1228.385,182.152,-54.493,-177.578,5.900,148.327
C04417=1228.389,181.903,-54.470,-177.580,5.898,148.327
C04418=1228.393,181.654,-54.447,-177.583,5.896,148.328
C04419=1228.398,181.406,-54.425,-177.585,5.895,148.328
C04420=1228.403,181.157,-54.402,-177.588,5.894,148.329
C04421=1228.408,180.908,-54.378,-177.590,5.893,148.329
C04422=1228.412,180.658,-54.356,-177.593,5.891,148.330
C04423=1228.417,180.410,-54.333,-177.596,5.889,148.330
C04424=1228.421,180.161,-54.311,-177.598,5.889,148.330
C04425=1228.426,179.912,-54.288,-177.601,5.887,148.331
C04426=1228.431,179.664,-54.266,-177.603,5.885,148.331
C04427=1228.435,179.415,-54.242,-177.606,5.884,148.332
C04428=1228.440,179.165,-54.220,-177.609,5.882,148.332
C04429=1228.444,178.916,-54.197,-177.611,5.881,148.333
C04430=1228.449,178.668,-54.175,-177.613,5.879,148.333
C04431=1228.454,178.419,-54.152,-177.616,5.878,148.333
C04432=1228.458,178.169,-54.130,-177.619,5.877,148.334
C04433=1228.464,177.921,-54.107,-177.621,5.875,148.334
C04434=1228.468,177.672,-54.084,-177.624,5.873,148.335
C04435=1228.473,177.423,-54.061,-177.626,5.872,148.335
C04436=1228.477,177.175,-54.039,-177.629,5.871,148.336
C04437=1228.481,176.925,-54.017,-177.631,5.870,148.336
C04438=1228.486,176.676,-53.994,-177.634,5.868,148.336
C04439=1228.491,176.428,-53.972,-177.637,5.866,148.337
C04440=1228.496,176.179,-53.949,-177.639,5.865,148.337
C04441=1228.500,175.929,-53.926,-177.642,5.864,148.338
C04442=1228.506,175.680,-53.904,-177.644,5.863,148.338
C04443=1228.509,175.431,-53.881,-177.647,5.861,148.339
C04444=1228.514,175.182,-53.859,-177.650,5.859,148.339
C04445=1228.519,174.934,-53.836,-177.652,5.858,148.339
C04446=1228.523,174.684,-53.814,-177.654,5.856,148.340
C04447=1228.528,174.435,-53.791,-177.657,5.856,148.340
C04448=1228.533,174.187,-53.769,-177.660,5.854,148.341
C04449=1228.537,173.937,-53.747,-177.662,5.853,148.341
C04450=1228.542,173.689,-53.724,-177.664,5.851,148.341
C04451=1228.547,173.440,-53.702,-177.668,5.850,148.342
C04452=1228.551,173.190,-53.680,-177.670,5.849,148.342
C04453=1228.556,172.942,-53.657,-177.672,5.847,148.343
C04454=1228.561,172.693,-53.635,-177.675,5.846,148.343
C04455=1228.565,172.444,-53.613,-177.677,5.844,148.344
C04456=1228.570,172.195,-53.590,-177.680,5.842,148.344
C04457=1228.574,171.946,-53.568,-177.683,5.842,148.345
C04458=1228.579,171.697,-53.546,-177.685,5.840,148.345
C04459=1228.584,171.448,-53.523,-177.687,5.839,148.345
C04460=1228.589,171.199,-53.501,-177.690,5.837,148.346
C04461=1228.593,170.950,-53.479,-177.693,5.836,148.346
C04462=1228.597,170.701,-53.457,-177.695,5.835,148.347
C04463=1228.603,170.452,-53.434,-177.697,5.834,148.347
C04464=1228.607,170.203,-53.412,-177.701,5.832,148.348
C04465=1228.612,169.954,-53.390,-177.703,5.830,148.348
C04466=1228.617,169.705,-53.368,-177.705,5.829,148.348
C04467=1228.621,169.457,-53.345,-177.709,5.828,148.349
C04468=1228.626,169.207,-53.323,-177.711,5.827,148.349
C04469=1228.631,168.959,-53.302,-177.713,5.825,148.350
C04470=1228.635,168.709,-53.280,-177.715,5.824,148.350
C04471=1228.640,168.461,-53.257,-177.718,5.822,148.351
C04472=1228.645,168.211,-53.235,-177.721,5.821,148.351
C04473=1228.649,167.963,-53.213,-177.723,5.820,148.352
C04474=1228.653,167.714,-53.191,-177.726,5.818,148.352
C04475=1228.659,167.465,-53.169,-177.728,5.817,148.352
C04476=1228.663,167.216,-53.147,-177.731,5.815,148.353
C04477=1228.668,166.966,-53.125,-177.734,5.815,148.353
C04478=1228.673,166.718,-53.103,-177.736,5.813,148.354
C04479=1228.677,166.468,-53.081,-177.738,5.812,148.354
C04480=1228.682,166.220,-53.059,-177.742,5.810,148.355
C04481=1228.687,165.971,-53.037,-177.744,5.809,148.355
C04482=1228.692,165.721,-53.015,-177.746,5.807,148.356
C04483=1228.696,165.473,-52.993,-177.749,5.807,148.356
C04484=1228.701,165.223,-52.971,-177.752,5.805,148.357
C04485=1228.705,164.975,-52.949,-177.754,5.803,148.357
C04486=1228.709,164.726,-52.927,-177.757,5.802,148.358
C04487=1228.714,164.477,-52.905,-177.760,5.801,148.358
C04488=1228.719,164.228,-52.883,-177.762,5.800,148.358
C04489=1228.723,163.979,-52.861,-177.765,5.798,148.359
C04490=1228.729,163.729,-52.839,-177.767,5.797,148.359
C04491=1228.734,163.480,-52.818,-177.770,5.795,148.360
C04492=1228.738,163.231,-52.796,-177.772,5.795,148.360
C04493=1228.743,162.982,-52.774,-177.775,5.793,148.361
C04494=1228.748,162.734,-52.752,-177.777,5.792,148.361
C04495=1228.752,162.484,-52.730,-177.780,5.790,148.362
C04496=1228.757,162.236,-52.708,-177.782,5.789,148.362
C04497=1228.761,161.986,-52.686,-177.785,5.788,148.363
C04498=1228.766,161.738,-52.665,-177.787,5.787,148.363
C04499=1228.770,161.488,-52.643,-177.790,5.785,148.363
C04500=1228.775,161.240,-52.621,-177.793,5.784,148.364
C04501=1228.780,160.991,-52.599,-177.795,5.782,148.364
C04502=1228.785,160.741,-52.578,-177.797,5.781,148.365
C04503=1228.789,160.493,-52.556,-177.801,5.780,148.365
C04504=1228.794,160.243,-52.534,-177.803,5.779,148.366
C04505=1228.799,159.974,-52.510,-177.806,5.777,148.366
C04506=1228.804,159.705,-52.487,-177.808,5.776,148.367
C04507=1228.809,159.436,-52.464,-177.811,5.775,148.367
C04508=1228.814,159.167,-52.440,-177.814,5.773,148.368
C04509=1228.819,158.918,-52.419,-177.817,5.772,148.368
C04510=1228.823,158.669,-52.398,-177.819,5.771,148.369
C04511=1228.828,158.420,-52.376,-177.822,5.769,148.369
C04512=1228.833,158.172,-52.354,-177.824,5.768,148.370
C04513=1228.837,157.922,-52.333,-177.827,5.766,148.370
C04514=1228.842,157.673,-52.311,-177.829,5.766,148.371
C04515=1228.847,157.425,-52.289,-177.832,5.765,148.371
C04516=1228.851,157.175,-52.267,-177.834,5.763,148.371
C04517=1228.856,156.926,-52.246,-177.837,5.762,148.372
C04518=1228.861,156.677,-52.225,-177.839,5.760,148.372
C04519=1228.866,156.428,-52.203,-177.842,5.759,148.373
C04520=1228.871,156.179,-52.182,-177.845,5.758,148.373
C04521=1228.876,155.930,-52.160,-177.847,5.757,148.374
C04522=1228.879,155.681,-52.139,-177.850,5.755,148.374
C04523=1228.884,155.432,-52.118,-177.852,5.754,148.375
C04524=1228.889,155.183,-52.096,-177.855,5.753,148.375
C04525=1228.893,154.934,-52.074,-177.857,5.752,148.376
C04526=1228.899,154.685,-52.053,-177.860,5.750,148.376
C04527=1228.904,154.436,-52.031,-177.863,5.749,148.377
C04528=1228.909,154.187,-52.010,-177.865,5.748,148.377
C04529=1228.912,153.938,-51.989,-177.867,5.747,148.377
C04530=1228.917,153.689,-51.967,-177.870,5.745,148.378
C04531=1228.922,153.440,-51.946,-177.873,5.744,148.378
C04532=1228.927,153.191,-51.925,-177.875,5.744,148.379
C04533=1228.932,152.941,-51.903,-177.878,5.742,148.379
C04534=1228.936,152.693,-51.882,-177.880,5.741,148.380
C04535=1228.941,152.443,-51.861,-177.883,5.739,148.380
C04536=1228.945,152.194,-51.839,-177.885,5.738,148.381
C04537=1228.950,151.945,-51.818,-177.888,5.737,148.381
C04538=1228.955,151.696,-51.796,-177.890,5.736,148.382
C04539=1228.960,151.447,-51.776,-177.894,5.734,148.382
C04540=1228.965,151.199,-51.754,-177.896,5.733,148.383
C04541=1228.969,150.949,-51.733,-177.898,5.732,148.383
C04542=1228.974,150.700,-51.711,-177.901,5.731,148.384
C04543=1228.979,150.451,-51.691,-177.903,5.730,148.384
C04544=1228.983,150.202,-51.669,-177.906,5.728,148.385
C04545=1228.988,149.953,-51.648,-177.908,5.727,148.385
C04546=1228.993,149.704,-51.626,-177.911,5.726,148.386
C04547=1228.997,149.455,-51.606,-177.914,5.725,148.386
C04548=1229.002,149.206,-51.585,-177.916,5.723,148.387
C04549=1229.007,148.957,-51.563,-177.919,5.722,148.387
C04550=1229.011,148.707,-51.543,-177.921,5.721,148.388
C04551=1229.016,148.459,-51.521,-177.924,5.720,148.388
C04552=1229.021,148.209,-51.500,-177.926,5.719,148.389
C04553=1229.026,147.961,-51.480,-177.929,5.717,148.389
C04554=1229.030,147.712,-51.458,-177.931,5.716,148.390
C04555=1229.035,147.462,-51.437,-177.934,5.715,148.390
C04556=1229.040,147.213,-51.416,-177.937,5.714,148.391
C04557=1229.044,146.964,-51.394,-177.939,5.713,148.391
C04558=1229.050,146.715,-51.373,-177.942,5.712,148.392
C04559=1229.054,146.466,-51.353,-177.944,5.711,148.392
C04560=1229.059,146.217,-51.331,-177.947,5.709,148.393
C04561=1229.063,145.968,-51.310,-177.949,5.708,148.393
C04562=1229.068,145.719,-51.290,-177.951,5.707,148.393
C04563=1229.073,145.469,-51.269,-177.955,5.706,148.394
C04564=1229.077,145.221,-51.248,-177.957,5.705,148.394
C04565=1229.082,144.972,-51.227,-177.960,5.703,148.395
C04566=1229.087,144.723,-51.206,-177.962,5.702,148.395
C04567=1229.092,144.474,-51.185,-177.965,5.701,148.396
C04568=1229.096,144.224,-51.163,-177.967,5.700,148.396
C04569=1229.101,143.975,-51.143,-177.970,5.699,148.397
C04570=1229.106,143.726,-51.122,-177.972,5.697,148.397
C04571=1229.110,143.477,-51.102,-177.975,5.697,148.398
C04572=1229.115,143.228,-51.081,-177.977,5.696,148.398
C04573=1229.120,142.979,-51.060,-177.980,5.694,148.399
C04574=1229.125,142.730,-51.039,-177.982,5.693,148.399
C04575=1229.129,142.481,-51.018,-177.985,5.691,148.400
C04576=1229.134,142.232,-50.997,-177.988,5.691,148.400
C04577=1229.139,141.983,-50.977,-177.990,5.690,148.401
C04578=1229.143,141.733,-50.956,-177.993,5.688,148.401
C04579=1229.148,141.484,-50.935,-177.995,5.687,148.402
C04580=1229.153,141.235,-50.913,-177.998,5.686,148.402
C04581=1229.157,140.987,-50.893,-178.000,5.685,148.403
C04582=1229.162,140.737,-50.872,-178.003,5.684,148.403
C04583=1229.167,140.488,-50.852,-178.006,5.682,148.404
C04584=1229.172,140.239,-50.831,-178.008,5.682,148.404
C04585=1229.176,139.990,-50.810,-178.011,5.680,148.405
C04586=1229.182,139.741,-50.789,-178.014,5.679,148.405
C04587=1229.186,139.492,-50.769,-178.016,5.678,148.406
C04588=1229.191,139.243,-50.748,-178.019,5.677,148.407
C04589=1229.196,138.994,-50.728,-178.021,5.676,148.407
C04590=1229.201,138.744,-50.707,-178.023,5.675,148.408
C04591=1229.205,138.495,-50.686,-178.026,5.673,148.408
C04592=1229.210,138.247,-50.666,-178.029,5.673,148.409
C04593=1229.215,137.997,-50.645,-178.031,5.672,148.409
C04594=1229.219,137.748,-50.625,-178.034,5.670,148.410
C04595=1229.224,137.499,-50.604,-178.036,5.669,148.410
C04596=1229.229,137.250,-50.583,-178.039,5.668,148.411
C04597=1229.233,137.001,-50.563,-178.041,5.667,148.411
C04598=1229.238,136.752,-50.542,-178.044,5.666,148.412
C04599=1229.243,136.503,-50.522,-178.047,5.664,148.412
C04600=1229.248,136.254,-50.501,-178.049,5.664,148.413
C04601=1229.253,136.004,-50.481,-178.051,5.663,148.413
C04602=1229.257,135.755,-50.461,-178.055,5.661,148.414
C04603=1229.262,135.506,-50.440,-178.057,5.660,148.414
C04604=1229.267,135.257,-50.419,-178.059,5.660,148.415
C04605=1229.271,135.008,-50.399,-178.062,5.658,148.415
C04606=1229.276,134.759,-50.378,-178.065,5.657,148.416
C04607=1229.281,134.510,-50.358,-178.067,5.656,148.416
C04608=1229.285,134.261,-50.337,-178.070,5.655,148.417
C04609=1229.291,133.992,-50.316,-178.072,5.654,148.417
C04610=1229.296,133.723,-50.293,-178.075,5.652,148.418
C04611=1229.301,133.454,-50.272,-178.078,5.652,148.418
C04612=1229.306,133.186,-50.249,-178.080,5.650,148.419
C04613=1229.310,132.937,-50.229,-178.083,5.649,148.419
C04614=1229.316,132.687,-50.209,-178.086,5.648,148.420
C04615=1229.320,132.438,-50.188,-178.088,5.647,148.420
C04616=1229.325,132.189,-50.168,-178.091,5.646,148.421
C04617=1229.329,131.940,-50.148,-178.094,5.644,148.421
C04618=1229.335,131.690,-50.127,-178.096,5.644,148.422
C04619=1229.339,131.441,-50.107,-178.098,5.643,148.422
C04620=1229.344,131.193,-50.087,-178.101,5.641,148.423
C04621=1229.349,130.944,-50.067,-178.104,5.640,148.423
C04622=1229.354,130.694,-50.046,-178.106,5.640,148.424
C04623=1229.359,130.445,-50.026,-178.109,5.638,148.424
C04624=1229.363,130.196,-50.006,-178.111,5.637,148.425
C04625=1229.368,129.947,-49.986,-178.113,5.636,148.425
C04626=1229.372,129.698,-49.966,-178.116,5.635,148.426
C04627=1229.377,129.449,-49.945,-178.119,5.634,148.427
C04628=1229.382,129.199,-49.925,-178.121,5.633,148.427
C04629=1229.387,128.951,-49.905,-178.124,5.632,148.428
C04630=1229.392,128.702,-49.885,-178.127,5.631,148.428
C04631=1229.396,128.452,-49.865,-178.129,5.630,148.429
C04632=1229.401,128.203,-49.845,-178.131,5.629,148.429
C04633=1229.406,127.953,-49.824,-178.135,5.628,148.430
C04634=1229.411,127.704,-49.804,-178.137,5.627,148.430
C04635=1229.415,127.456,-49.784,-178.139,5.626,148.431
C04636=1229.420,127.206,-49.764,-178.142,5.624,148.431
C04637=1229.425,126.958,-49.744,-178.145,5.623,148.432
C04638=1229.430,126.708,-49.724,-178.147,5.622,148.432
C04639=1229.434,126.459,-49.704,-178.149,5.622,148.433
C04640=1229.439,126.210,-49.684,-178.152,5.620,148.434
C04641=1229.444,125.960,-49.663,-178.155,5.619,148.434
C04642=1229.449,125.711,-49.644,-178.157,5.619,148.435
C04643=1229.454,125.463,-49.624,-178.160,5.617,148.435
C04644=1229.458,125.213,-49.604,-178.162,5.616,148.436
C04645=1229.463,124.964,-49.584,-178.165,5.615,148.436
C04646=1229.468,124.714,-49.564,-178.168,5.614,148.437
C04647=1229.472,124.466,-49.544,-178.170,5.613,148.437
C04648=1229.477,124.217,-49.524,-178.172,5.612,148.438
C04649=1229.482,123.968,-49.504,-178.175,5.612,148.438
C04650=1229.487,123.718,-49.484,-178.178,5.610,148.439
C04651=1229.491,123.469,-49.464,-178.180,5.609,148.439
C04652=1229.496,123.220,-49.444,-178.182,5.608,148.440
C04653=1229.501,122.971,-49.424,-178.185,5.608,148.440
C04654=1229.506,122.722,-49.405,-178.188,5.606,148.441
C04655=1229.510,122.472,-49.385,-178.190,5.605,148.441
C04656=1229.515,122.223,-49.364,-178.193,5.605,148.442
C04657=1229.520,121.974,-49.345,-178.196,5.603,148.442
C04658=1229.525,121.725,-49.326,-178.198,5.602,148.443
C04659=1229.529,121.476,-49.305,-178.200,5.601,148.443
C04660=1229.534,121.226,-49.285,-178.203,5.601,148.444
C04661=1229.539,120.978,-49.265,-178.206,5.599,148.445
C04662=1229.544,120.729,-49.246,-178.208,5.598,148.445
C04663=1229.549,120.479,-49.226,-178.211,5.597,148.446
C04664=1229.553,120.229,-49.207,-178.213,5.596,148.446
C04665=1229.558,119.981,-49.187,-178.216,5.595,148.447
C04666=1229.563,119.732,-49.167,-178.219,5.594,148.447
C04667=1229.568,119.482,-49.147,-178.221,5.593,148.448
C04668=1229.573,119.234,-49.127,-178.224,5.592,148.448
C04669=1229.578,118.984,-49.108,-178.226,5.591,148.449
C04670=1229.582,118.735,-49.088,-178.229,5.590,148.450
C04671=1229.587,118.485,-49.068,-178.231,5.590,148.450
C04672=1229.592,118.237,-49.048,-178.234,5.588,148.451
C04673=1229.596,117.988,-49.029,-178.237,5.587,148.451
C04674=1229.601,117.738,-49.010,-178.239,5.586,148.452
C04675=1229.606,117.489,-48.990,-178.241,5.586,148.452
C04676=1229.611,117.240,-48.970,-178.245,5.584,148.453
C04677=1229.615,116.991,-48.950,-178.247,5.583,148.453
C04678=1229.621,116.742,-48.931,-178.249,5.583,148.454
C04679=1229.626,116.492,-48.911,-178.251,5.582,148.454
C04680=1229.630,116.243,-48.892,-178.254,5.581,148.455
C04681=1229.635,115.994,-48.873,-178.257,5.580,148.456
C04682=1229.639,115.745,-48.853,-178.259,5.579,148.456
C04683=1229.644,115.496,-48.833,-178.262,5.578,148.457
C04684=1229.649,115.247,-48.814,-178.264,5.577,148.457
C04685=1229.654,114.997,-48.794,-178.267,5.576,148.458
C04686=1229.659,114.748,-48.774,-178.270,5.575,148.458
C04687=1229.663,114.499,-48.756,-178.272,5.574,148.459
C04688=1229.668,114.249,-48.736,-178.275,5.573,148.459
C04689=1229.673,114.000,-48.716,-178.277,5.572,148.460
C04690=1229.678,113.751,-48.697,-178.280,5.571,148.460
C04691=1229.683,113.501,-48.677,-178.282,5.570,148.461
C04692=1229.687,113.253,-48.658,-178.285,5.569,148.461
C04693=1229.692,113.004,-48.638,-178.287,5.569,148.462
C04694=1229.697,112.754,-48.619,-178.290,5.567,148.463
C04695=1229.702,112.505,-48.599,-178.292,5.566,148.463
C04696=1229.707,112.256,-48.580,-178.295,5.566,148.464
C04697=1229.712,112.007,-48.561,-178.297,5.565,148.464
C04698=1229.716,111.758,-48.541,-178.300,5.563,148.465
C04699=1229.721,111.508,-48.522,-178.303,5.563,148.465
C04700=1229.726,111.260,-48.503,-178.305,5.562,148.466
C04701=1229.730,111.010,-48.483,-178.308,5.561,148.467
C04702=1229.736,110.761,-48.464,-178.310,5.560,148.467
C04703=1229.740,110.512,-48.444,-178.313,5.559,148.468
C04704=1229.744,110.262,-48.425,-178.316,5.558,148.468
C04705=1229.750,110.013,-48.407,-178.318,5.557,148.469
C04706=1229.755,109.763,-48.387,-178.320,5.556,148.469
C04707=1229.759,109.515,-48.368,-178.323,5.556,148.470
C04708=1229.764,109.265,-48.349,-178.326,5.554,148.471
C04709=1229.770,109.016,-48.329,-178.328,5.553,148.471
C04710=1229.774,108.767,-48.310,-178.331,5.553,148.472
C04711=1229.779,108.518,-48.291,-178.333,5.552,148.472
C04712=1229.784,108.269,-48.271,-178.336,5.551,148.473
C04713=1229.789,108.000,-48.250,-178.339,5.550,148.473
C04714=1229.794,107.732,-48.231,-178.341,5.549,148.474
C04715=1229.799,107.463,-48.210,-178.345,5.548,148.475
C04716=1229.804,107.195,-48.189,-178.347,5.547,148.475
C04717=1229.809,106.946,-48.169,-178.349,5.546,148.476
C04718=1229.814,106.696,-48.151,-178.352,5.546,148.476
C04719=1229.818,106.447,-48.132,-178.355,5.545,148.477
C04720=1229.824,106.198,-48.112,-178.357,5.543,148.477
C04721=1229.828,105.949,-48.093,-178.360,5.542,148.478
C04722=1229.833,105.700,-48.074,-178.362,5.542,148.479
C04723=1229.837,105.450,-48.056,-178.365,5.541,148.479
C04724=1229.843,105.201,-48.037,-178.367,5.540,148.480
C04725=1229.848,104.952,-48.017,-178.370,5.539,148.480
C04726=1229.852,104.703,-47.998,-178.373,5.538,148.481
C04727=1229.857,104.453,-47.979,-178.375,5.537,148.481
C04728=1229.862,104.204,-47.961,-178.378,5.537,148.482
C04729=1229.867,103.955,-47.941,-178.380,5.536,148.482
C04730=1229.871,103.705,-47.923,-178.382,5.535,148.483
C04731=1229.876,103.456,-47.903,-178.386,5.534,148.484
C04732=1229.881,103.207,-47.885,-178.388,5.533,148.484
C04733=1229.886,102.958,-47.865,-178.390,5.532,148.485
C04734=1229.890,102.709,-47.847,-178.393,5.531,148.485
C04735=1229.896,102.460,-47.828,-178.395,5.530,148.486
C04736=1229.900,102.210,-47.809,-178.398,5.530,148.486
C04737=1229.905,101.961,-47.790,-178.401,5.528,148.487
C04738=1229.909,101.712,-47.771,-178.403,5.527,148.488
C04739=1229.915,101.462,-47.752,-178.406,5.527,148.488
C04740=1229.919,101.213,-47.733,-178.408,5.526,148.489
C04741=1229.924,100.964,-47.714,-178.410,5.525,148.489
C04742=1229.929,100.715,-47.696,-178.413,5.525,148.490
C04743=1229.934,100.465,-47.676,-178.416,5.523,148.491
C04744=1229.939,100.217,-47.658,-178.418,5.522,148.491
C04745=1229.944,99.967,-47.639,-178.421,5.522,148.492
C04746=1229.948,99.718,-47.620,-178.424,5.521,148.492
C04747=1229.953,99.468,-47.601,-178.426,5.520,148.493
C04748=1229.958,99.219,-47.582,-178.428,5.519,148.493
C04749=1229.963,98.970,-47.564,-178.431,5.519,148.494
C04750=1229.968,98.721,-47.545,-178.434,5.517,148.495
C04751=1229.973,98.471,-47.527,-178.436,5.516,148.495
C04752=1229.978,98.223,-47.507,-178.439,5.516,148.496
C04753=1229.982,97.973,-47.489,-178.441,5.515,148.496
C04754=1229.987,97.724,-47.470,-178.444,5.514,148.497
C04755=1229.992,97.474,-47.451,-178.446,5.514,148.497
C04756=1229.997,97.225,-47.433,-178.449,5.513,148.498
C04757=1230.002,96.976,-47.414,-178.452,5.511,148.498
C04758=1230.006,96.727,-47.395,-178.454,5.511,148.499
C04759=1230.011,96.477,-47.377,-178.457,5.510,148.500
C04760=1230.016,96.229,-47.358,-178.459,5.509,148.500
C04761=1230.021,95.979,-47.340,-178.462,5.508,148.501
C04762=1230.025,95.730,-47.321,-178.464,5.508,148.501
C04763=1230.031,95.481,-47.302,-178.467,5.507,148.502
C04764=1230.035,95.231,-47.284,-178.469,5.505,148.503
C04765=1230.040,94.982,-47.265,-178.472,5.505,148.503
C04766=1230.046,94.733,-47.247,-178.475,5.504,148.504
C04767=1230.050,94.483,-47.228,-178.477,5.504,148.504
C04768=1230.054,94.234,-47.210,-178.479,5.503,148.505
C04769=1230.060,93.985,-47.191,-178.482,5.502,148.506
C04770=1230.064,93.736,-47.172,-178.485,5.501,148.506
C04771=1230.069,93.486,-47.154,-178.487,5.501,148.507
C04772=1230.075,93.237,-47.135,-178.489,5.500,148.507
C04773=1230.079,92.988,-47.116,-178.493,5.498,148.508
C04774=1230.084,92.738,-47.098,-178.495,5.498,148.509
C04775=1230.089,92.489,-47.080,-178.497,5.497,148.509
C04776=1230.093,92.240,-47.061,-178.500,5.496,148.510
C04777=1230.098,91.991,-47.043,-178.503,5.496,148.510
C04778=1230.103,91.741,-47.025,-178.505,5.495,148.511
C04779=1230.108,91.492,-47.007,-178.507,5.494,148.511
C04780=1230.113,91.243,-46.987,-178.510,5.494,148.512
C04781=1230.118,90.993,-46.969,-178.513,5.493,148.513
C04782=1230.123,90.744,-46.951,-178.515,5.491,148.513
C04783=1230.127,90.496,-46.932,-178.518,5.491,148.514
C04784=1230.131,90.246,-46.914,-178.521,5.490,148.514
C04785=1230.137,89.996,-46.896,-178.523,5.489,148.515
C04786=1230.142,89.747,-46.878,-178.525,5.488,148.515
C04787=1230.147,89.498,-46.860,-178.528,5.488,148.516
C04788=1230.151,89.249,-46.841,-178.531,5.487,148.517
C04789=1230.156,89.000,-46.823,-178.533,5.487,148.517
C04790=1230.162,88.750,-46.804,-178.535,5.486,148.518
C04791=1230.166,88.501,-46.786,-178.538,5.485,148.518
C04792=1230.171,88.251,-46.768,-178.541,5.484,148.519
C04793=1230.176,88.002,-46.750,-178.544,5.483,148.520
C04794=1230.180,87.753,-46.731,-178.546,5.482,148.520
C04795=1230.185,87.504,-46.713,-178.548,5.481,148.521
C04796=1230.191,87.255,-46.694,-178.551,5.481,148.521
C04797=1230.195,87.005,-46.676,-178.554,5.480,148.522
C04798=1230.200,86.756,-46.658,-178.556,5.479,148.523
C04799=1230.205,86.506,-46.640,-178.558,5.479,148.523
C04800=1230.210,86.257,-46.622,-178.561,5.478,148.524
C04801=1230.215,86.008,-46.604,-178.564,5.477,148.525
C04802=1230.219,85.758,-46.586,-178.566,5.476,148.525
C04803=1230.224,85.510,-46.567,-178.568,5.476,148.526
C04804=1230.229,85.260,-46.549,-178.572,5.474,148.526
C04805=1230.234,85.011,-46.531,-178.574,5.474,148.527
C04806=1230.239,84.762,-46.513,-178.576,5.473,148.527
C04807=1230.243,84.512,-46.494,-178.579,5.472,148.528
C04808=1230.248,84.263,-46.476,-178.582,5.472,148.529
C04809=1230.253,84.014,-46.458,-178.584,5.471,148.529
C04810=1230.258,83.764,-46.440,-178.586,5.470,148.530
C04811=1230.263,83.515,-46.422,-178.589,5.470,148.530
C04812=1230.268,83.266,-46.404,-178.592,5.469,148.531
C04813=1230.273,83.017,-46.386,-178.594,5.468,148.532
C04814=1230.277,82.767,-46.368,-178.597,5.468,148.532
C04815=1230.282,82.518,-46.350,-178.599,5.467,148.533
C04816=1230.287,82.269,-46.332,-178.602,5.466,148.533
C04817=1230.292,82.000,-46.313,-178.605,5.465,148.534
C04818=1230.298,81.732,-46.294,-178.607,5.464,148.535
C04819=1230.303,81.463,-46.275,-178.610,5.464,148.535
C04820=1230.308,81.195,-46.255,-178.613,5.463,148.536
C04821=1230.313,80.946,-46.237,-178.615,5.462,148.537
C04822=1230.318,80.697,-46.219,-178.618,5.462,148.537
C04823=1230.322,80.447,-46.201,-178.620,5.461,148.538
C04824=1230.328,80.198,-46.184,-178.623,5.460,148.538
C04825=1230.333,79.949,-46.166,-178.625,5.460,148.539
C04826=1230.338,79.699,-46.148,-178.629,5.458,148.540
C04827=1230.342,79.449,-46.130,-178.631,5.458,148.540
C04828=1230.347,79.200,-46.112,-178.633,5.457,148.541
C04829=1230.352,78.951,-46.094,-178.636,5.456,148.541
C04830=1230.357,78.702,-46.076,-178.639,5.456,148.542
C04831=1230.362,78.452,-46.058,-178.641,5.455,148.543
C04832=1230.367,78.203,-46.040,-178.643,5.454,148.543
C04833=1230.372,77.954,-46.022,-178.646,5.453,148.544
C04834=1230.377,77.705,-46.005,-178.649,5.453,148.545
C04835=1230.381,77.455,-45.987,-178.651,5.452,148.545
C04836=1230.387,77.206,-45.969,-178.654,5.452,148.546
C04837=1230.391,76.957,-45.952,-178.656,5.451,148.546
C04838=1230.396,76.708,-45.934,-178.659,5.450,148.547
C04839=1230.401,76.458,-45.916,-178.661,5.449,148.548
C04840=1230.406,76.209,-45.899,-178.664,5.449,148.548
C04841=1230.411,75.959,-45.881,-178.666,5.448,148.549
C04842=1230.416,75.710,-45.863,-178.669,5.447,148.549
C04843=1230.421,75.461,-45.845,-178.671,5.447,148.550
C04844=1230.425,75.212,-45.828,-178.674,5.446,148.551
C04845=1230.430,74.962,-45.810,-178.676,5.446,148.551
C04846=1230.434,74.713,-45.792,-178.679,5.445,148.552
C04847=1230.440,74.463,-45.774,-178.681,5.444,148.552
C04848=1230.444,74.214,-45.756,-178.684,5.443,148.553
C04849=1230.449,73.964,-45.738,-178.686,5.443,148.554
C04850=1230.454,73.715,-45.722,-178.689,5.442,148.554
C04851=1230.459,73.466,-45.704,-178.692,5.442,148.555
C04852=1230.464,73.217,-45.686,-178.694,5.441,148.555
C04853=1230.469,72.967,-45.669,-178.697,5.440,148.556
C04854=1230.474,72.718,-45.651,-178.699,5.440,148.557
C04855=1230.479,72.469,-45.634,-178.702,5.439,148.557
C04856=1230.484,72.220,-45.616,-178.704,5.438,148.558
C04857=1230.489,71.970,-45.598,-178.707,5.438,148.559
C04858=1230.494,71.721,-45.581,-178.709,5.437,148.559
C04859=1230.498,71.472,-45.564,-178.712,5.436,148.560
C04860=1230.503,71.223,-45.546,-178.714,5.436,148.561
C04861=1230.508,70.973,-45.528,-178.717,5.435,148.561
C04862=1230.513,70.724,-45.510,-178.720,5.434,148.562
C04863=1230.518,70.474,-45.494,-178.722,5.433,148.562
C04864=1230.523,70.225,-45.476,-178.724,5.433,148.563
C04865=1230.528,69.975,-45.459,-178.727,5.432,148.564
C04866=1230.533,69.726,-45.441,-178.730,5.432,148.564
C04867=1230.537,69.477,-45.424,-178.732,5.431,148.565
C04868=1230.542,69.227,-45.406,-178.735,5.431,148.566
C04869=1230.547,68.978,-45.389,-178.737,5.430,148.566
C04870=1230.551,68.729,-45.371,-178.740,5.429,148.567
C04871=1230.557,68.479,-45.354,-178.742,5.428,148.567
C04872=1230.562,68.230,-45.336,-178.745,5.428,148.568
C04873=1230.566,67.980,-45.319,-178.748,5.427,148.569
C04874=1230.572,67.732,-45.302,-178.750,5.427,148.569
C04875=1230.577,67.482,-45.284,-178.752,5.426,148.570
C04876=1230.581,67.233,-45.267,-178.755,5.425,148.570
C04877=1230.586,66.983,-45.250,-178.758,5.425,148.571
C04878=1230.591,66.734,-45.233,-178.760,5.424,148.572
C04879=1230.596,66.485,-45.215,-178.763,5.423,148.572
C04880=1230.601,66.235,-45.198,-178.766,5.423,148.573
C04881=1230.606,65.986,-45.180,-178.768,5.422,148.574
C04882=1230.610,65.736,-45.163,-178.770,5.421,148.574
C04883=1230.615,65.486,-45.146,-178.773,5.421,148.575
C04884=1230.620,65.238,-45.129,-178.776,5.420,148.576
C04885=1230.625,64.988,-45.112,-178.778,5.420,148.576
C04886=1230.631,64.739,-45.094,-178.781,5.419,148.577
C04887=1230.635,64.490,-45.077,-178.783,5.418,148.577
C04888=1230.640,64.240,-45.060,-178.786,5.417,148.578
C04889=1230.644,63.991,-45.043,-178.788,5.417,148.579
C04890=1230.649,63.741,-45.025,-178.791,5.416,148.579
C04891=1230.655,63.492,-45.008,-178.793,5.416,148.580
C04892=1230.660,63.243,-44.992,-178.796,5.415,148.581
C04893=1230.665,62.994,-44.974,-178.799,5.415,148.581
C04894=1230.669,62.744,-44.957,-178.801,5.414,148.582
C04895=1230.674,62.494,-44.940,-178.804,5.413,148.582
C04896=1230.679,62.245,-44.923,-178.806,5.412,148.583
C04897=1230.684,61.996,-44.905,-178.809,5.412,148.584
C04898=1230.689,61.747,-44.889,-178.811,5.411,148.584
C04899=1230.694,61.497,-44.871,-178.814,5.411,148.585
C04900=1230.698,61.248,-44.855,-178.816,5.410,148.585
C04901=1230.703,60.998,-44.837,-178.819,5.409,148.586
C04902=1230.708,60.750,-44.821,-178.821,5.409,148.587
C04903=1230.714,60.500,-44.803,-178.824,5.408,148.587
C04904=1230.718,60.250,-44.787,-178.827,5.407,148.588
C04905=1230.723,60.001,-44.769,-178.829,5.407,148.589
C04906=1230.728,59.752,-44.752,-178.831,5.407,148.589
C04907=1230.733,59.503,-44.735,-178.834,5.406,148.590
C04908=1230.738,59.253,-44.718,-178.836,5.406,148.591
C04909=1230.743,59.003,-44.701,-178.839,5.405,148.591
C04910=1230.748,58.754,-44.684,-178.841,5.404,148.592
C04911=1230.753,58.504,-44.667,-178.844,5.404,148.593
C04912=1230.758,58.256,-44.650,-178.847,5.403,148.593
C04913=1230.763,58.006,-44.633,-178.849,5.403,148.594
C04914=1230.767,57.757,-44.616,-178.852,5.402,148.595
C04915=1230.772,57.507,-44.600,-178.854,5.401,148.595
C04916=1230.778,57.258,-44.583,-178.857,5.401,148.596
C04917=1230.782,57.009,-44.566,-178.859,5.400,148.596
C04918=1230.787,56.759,-44.549,-178.862,5.399,148.597
C04919=1230.792,56.509,-44.532,-178.865,5.399,148.598
C04920=1230.798,56.260,-44.515,-178.867,5.398,148.598
C04921=1230.802,55.992,-44.497,-178.870,5.398,148.599
C04922=1230.807,55.724,-44.479,-178.873,5.397,148.600
C04923=1230.813,55.455,-44.461,-178.875,5.397,148.600
C04924=1230.818,55.187,-44.443,-178.878,5.396,148.601
C04925=1230.823,54.937,-44.426,-178.880,5.395,148.602
C04926=1230.828,54.688,-44.409,-178.883,5.395,148.602
C04927=1230.832,54.438,-44.392,-178.886,5.394,148.603
C04928=1230.838,54.189,-44.375,-178.888,5.394,148.604
C04929=1230.843,53.940,-44.359,-178.891,5.393,148.604
C04930=1230.847,53.690,-44.342,-178.894,5.392,148.605
C04931=1230.853,53.441,-44.325,-178.895,5.392,148.605
C04932=1230.857,53.192,-44.308,-178.898,5.392,148.606
C04933=1230.862,52.942,-44.292,-178.901,5.391,148.607
C04934=1230.868,52.693,-44.275,-178.903,5.391,148.607
C04935=1230.872,52.444,-44.258,-178.906,5.390,148.608
C04936=1230.877,52.194,-44.242,-178.908,5.390,148.609
C04937=1230.882,51.945,-44.225,-178.911,5.389,148.609
C04938=1230.887,51.695,-44.208,-178.914,5.388,148.610
C04939=1230.892,51.445,-44.192,-178.916,5.387,148.611
C04940=1230.897,51.196,-44.175,-178.918,5.387,148.611
C04941=1230.902,50.947,-44.158,-178.921,5.386,148.612
C04942=1230.906,50.697,-44.142,-178.924,5.386,148.613
C04943=1230.912,50.449,-44.126,-178.926,5.386,148.613
C04944=1230.917,50.199,-44.108,-178.928,5.385,148.614
C04945=1230.921,49.949,-44.092,-178.931,5.385,148.615
C04946=1230.926,49.700,-44.075,-178.934,5.384,148.615
C04947=1230.931,49.450,-44.059,-178.936,5.384,148.616
C04948=1230.936,49.201,-44.042,-178.939,5.383,148.617
C04949=1230.941,48.952,-44.026,-178.941,5.382,148.617
C04950=1230.946,48.702,-44.009,-178.944,5.382,148.618
C04951=1230.951,48.454,-43.993,-178.946,5.381,148.618
C04952=1230.956,48.203,-43.977,-178.949,5.380,148.619
C04953=1230.961,47.954,-43.960,-178.952,5.380,148.620
C04954=1230.966,47.705,-43.943,-178.954,5.380,148.620
C04955=1230.971,47.455,-43.927,-178.956,5.380,148.621
C04956=1230.975,47.206,-43.910,-178.959,5.379,148.622
C04957=1230.980,46.956,-43.894,-178.962,5.378,148.622
C04958=1230.986,46.707,-43.877,-178.964,5.378,148.623
C04959=1230.991,46.458,-43.861,-178.967,5.377,148.624
C04960=1230.995,46.208,-43.844,-178.969,5.376,148.624
C04961=1231.001,45.959,-43.829,-178.972,5.376,148.625
C04962=1231.005,45.710,-43.812,-178.974,5.375,148.626
C04963=1231.009,45.460,-43.795,-178.976,5.375,148.626
C04964=1231.015,45.211,-43.780,-178.979,5.375,148.627
C04965=1231.020,44.961,-43.762,-178.982,5.374,148.628
C04966=1231.025,44.712,-43.746,-178.984,5.374,148.628
C04967=1231.030,44.462,-43.730,-178.987,5.373,148.629
C04968=1231.035,44.213,-43.714,-178.990,5.373,148.630
C04969=1231.040,43.964,-43.697,-178.992,5.372,148.630
C04970=1231.044,43.714,-43.681,-178.995,5.372,148.631
C04971=1231.049,43.465,-43.665,-178.997,5.371,148.631
C04972=1231.054,43.215,-43.648,-178.999,5.371,148.632
C04973=1231.060,42.966,-43.632,-179.002,5.370,148.633
C04974=1231.064,42.716,-43.615,-179.004,5.370,148.633
C04975=1231.070,42.467,-43.599,-179.007,5.369,148.634
C04976=1231.074,42.217,-43.583,-179.010,5.369,148.635
C04977=1231.079,41.968,-43.567,-179.012,5.368,148.635
C04978=1231.084,41.718,-43.551,-179.015,5.367,148.636
C04979=1231.089,41.470,-43.535,-179.018,5.367,148.637
C04980=1231.094,41.219,-43.519,-179.020,5.367,148.637
C04981=1231.099,40.971,-43.502,-179.022,5.367,148.638
C04982=1231.104,40.721,-43.486,-179.025,5.366,148.639
C04983=1231.109,40.472,-43.470,-179.028,5.365,148.639
C04984=1231.114,40.222,-43.453,-179.030,5.365,148.640
C04985=1231.119,39.973,-43.438,-179.032,5.364,148.641
C04986=1231.123,39.723,-43.421,-179.035,5.363,148.641
C04987=1231.129,39.474,-43.405,-179.037,5.364,148.642
C04988=1231.133,39.225,-43.389,-179.040,5.363,148.643
C04989=1231.139,38.975,-43.373,-179.042,5.363,148.643
C04990=1231.143,38.726,-43.357,-179.045,5.362,148.644
C04991=1231.148,38.476,-43.341,-179.048,5.361,148.645
C04992=1231.153,38.227,-43.324,-179.050,5.361,148.645
C04993=1231.158,37.977,-43.309,-179.053,5.360,148.646
C04994=1231.163,37.728,-43.292,-179.055,5.361,148.647
C04995=1231.168,37.478,-43.276,-179.058,5.360,148.647
C04996=1231.174,37.229,-43.261,-179.060,5.359,148.648
C04997=1231.178,36.980,-43.244,-179.063,5.359,148.649
C04998=1231.183,36.730,-43.229,-179.066,5.358,148.649
C04999=1231.188,36.481,-43.212,-179.068,5.357,148.650
C05000=1231.193,36.231,-43.196,-179.070,5.357,148.650
C05001=1231.198,35.982,-43.180,-179.072,5.357,148.651
C05002=1231.203,35.732,-43.164,-179.075,5.357,148.652
C05003=1231.209,35.483,-43.149,-179.078,5.356,148.653
C05004=1231.213,35.234,-43.132,-179.080,5.355,148.653
C05005=1231.218,34.984,-43.116,-179.083,5.355,148.654
C05006=1231.223,34.734,-43.101,-179.086,5.354,148.655
C05007=1231.228,34.486,-43.085,-179.088,5.355,148.655
C05008=1231.232,34.235,-43.069,-179.090,5.354,148.656
C05009=1231.238,33.986,-43.053,-179.093,5.353,148.657
C05010=1231.243,33.737,-43.037,-179.096,5.353,148.657
C05011=1231.248,33.487,-43.021,-179.098,5.352,148.658
C05012=1231.253,33.238,-43.005,-179.101,5.352,148.659
C05013=1231.258,32.988,-42.989,-179.103,5.352,148.659
C05014=1231.262,32.739,-42.974,-179.106,5.351,148.660
C05015=1231.268,32.490,-42.958,-179.108,5.351,148.661
C05016=1231.272,32.240,-42.941,-179.111,5.350,148.661
C05017=1231.277,31.991,-42.926,-179.114,5.350,148.662
C05018=1231.283,31.741,-42.910,-179.116,5.349,148.662
C05019=1231.288,31.491,-42.894,-179.118,5.349,148.663
C05020=1231.292,31.243,-42.878,-179.120,5.349,148.664
C05021=1231.297,30.993,-42.862,-179.123,5.348,148.664
C05022=1231.302,30.743,-42.847,-179.126,5.347,148.665
C05023=1231.307,30.494,-42.831,-179.128,5.347,148.666
C05024=1231.312,30.244,-42.815,-179.131,5.346,148.667
C05025=1231.318,29.975,-42.798,-179.134,5.346,148.667
C05026=1231.323,29.707,-42.782,-179.137,5.346,148.668
C05027=1231.328,29.439,-42.765,-179.139,5.345,148.669
C05028=1231.334,29.170,-42.748,-179.141,5.345,148.669
C05029=1231.339,28.920,-42.732,-179.144,5.345,148.670
C05030=1231.344,28.671,-42.716,-179.147,5.344,148.671
C05031=1231.348,28.422,-42.701,-179.149,5.344,148.671
C05032=1231.353,28.172,-42.685,-179.152,5.343,148.672
C05033=1231.358,27.923,-42.669,-179.155,5.343,148.673
C05034=1231.364,27.673,-42.654,-179.157,5.343,148.674
C05035=1231.368,27.424,-42.638,-179.159,5.342,148.674
C05036=1231.373,27.174,-42.623,-179.162,5.342,148.675
C05037=1231.379,26.925,-42.607,-179.165,5.341,148.676
C05038=1231.384,26.675,-42.591,-179.167,5.341,148.676
C05039=1231.388,26.426,-42.575,-179.169,5.341,148.677
C05040=1231.393,26.177,-42.560,-179.172,5.340,148.677
C05041=1231.399,25.927,-42.544,-179.174,5.339,148.678
C05042=1231.403,25.678,-42.529,-179.177,5.339,148.679
C05043=1231.408,25.428,-42.513,-179.180,5.338,148.679
C05044=1231.413,25.179,-42.498,-179.182,5.339,148.680
C05045=1231.418,24.930,-42.483,-179.184,5.338,148.681
C05046=1231.423,24.680,-42.467,-179.187,5.337,148.681
C05047=1231.428,24.430,-42.451,-179.190,5.337,148.682
C05048=1231.433,24.181,-42.436,-179.192,5.336,148.683
C05049=1231.438,23.932,-42.420,-179.194,5.337,148.684
C05050=1231.443,23.682,-42.405,-179.197,5.336,148.684
C05051=1231.448,23.433,-42.390,-179.200,5.336,148.685
C05052=1231.453,23.183,-42.374,-179.202,5.335,148.686
C05053=1231.458,22.934,-42.358,-179.205,5.334,148.686
C05054=1231.462,22.684,-42.343,-179.207,5.335,148.687
C05055=1231.468,22.435,-42.327,-179.210,5.334,148.688
C05056=1231.473,22.185,-42.312,-179.212,5.334,148.688
C05057=1231.478,21.936,-42.297,-179.215,5.333,148.689
C05058=1231.483,21.686,-42.281,-179.217,5.333,148.690
C05059=1231.487,21.437,-42.266,-179.220,5.333,148.690
C05060=1231.493,21.187,-42.250,-179.222,5.332,148.691
C05061=1231.498,20.938,-42.235,-179.225,5.332,148.692
C05062=1231.503,20.688,-42.220,-179.227,5.331,148.692
C05063=1231.508,20.438,-42.204,-179.230,5.331,148.693
C05064=1231.513,20.189,-42.189,-179.232,5.331,148.694
C05065=1231.518,19.940,-42.174,-179.235,5.330,148.694
C05066=1231.523,19.691,-42.159,-179.238,5.330,148.695
C05067=1231.528,19.441,-42.143,-179.240,5.329,148.696
C05068=1231.533,19.191,-42.127,-179.242,5.329,148.696
C05069=1231.537,18.942,-42.112,-179.245,5.329,148.697
C05070=1231.543,18.692,-42.097,-179.248,5.328,148.698
C05071=1231.548,18.443,-42.083,-179.250,5.328,148.699
C05072=1231.553,18.194,-42.067,-179.253,5.327,148.699
C05073=1231.557,17.944,-42.052,-179.255,5.328,148.700
C05074=1231.563,17.694,-42.036,-179.258,5.327,148.701
C05075=1231.567,17.445,-42.021,-179.260,5.326,148.701
C05076=1231.573,17.195,-42.006,-179.263,5.326,148.702
C05077=1231.578,16.946,-41.991,-179.265,5.326,148.703
C05078=1231.583,16.697,-41.976,-179.268,5.326,148.703
C05079=1231.587,16.447,-41.960,-179.270,5.325,148.704
C05080=1231.593,16.197,-41.945,-179.273,5.325,148.705
C05081=1231.597,15.948,-41.930,-179.276,5.324,148.705
C05082=1231.603,15.698,-41.915,-179.278,5.324,148.706
C05083=1231.607,15.449,-41.900,-179.280,5.324,148.707
C05084=1231.613,15.199,-41.885,-179.283,5.323,148.707
C05085=1231.618,14.950,-41.870,-179.286,5.323,148.708
C05086=1231.623,14.701,-41.854,-179.288,5.323,148.709
C05087=1231.627,14.451,-41.839,-179.290,5.322,148.709
C05088=1231.632,14.201,-41.825,-179.293,5.322,148.710
C05089=1231.637,13.952,-41.809,-179.296,5.321,148.711
C05090=1231.642,13.703,-41.794,-179.298,5.322,148.712
C05091=1231.648,13.453,-41.779,-179.300,5.321,148.712
C05092=1231.652,13.204,-41.764,-179.303,5.321,148.713
C05093=1231.658,12.954,-41.749,-179.306,5.320,148.714
C05094=1231.663,12.705,-41.734,-179.308,5.320,148.714
C05095=1231.667,12.456,-41.719,-179.310,5.320,148.715
C05096=1231.673,12.206,-41.704,-179.313,5.319,148.716
C05097=1231.677,11.956,-41.689,-179.316,5.319,148.716
C05098=1231.683,11.706,-41.674,-179.318,5.319,148.717
C05099=1231.688,11.457,-41.659,-179.320,5.318,148.718
C05100=1231.692,11.207,-41.644,-179.323,5.318,148.718
C05101=1231.698,10.958,-41.629,-179.326,5.317,148.719
C05102=1231.703,10.708,-41.614,-179.328,5.318,148.720
C05103=1231.707,10.459,-41.599,-179.330,5.317,148.720
C05104=1231.713,10.209,-41.585,-179.333,5.317,148.721
C05105=1231.718,9.960,-41.570,-179.336,5.316,148.722
C05106=1231.723,9.711,-41.554,-179.338,5.316,148.722
C05107=1231.728,9.461,-41.540,-179.340,5.316,148.723
C05108=1231.732,9.212,-41.525,-179.343,5.315,148.724
C05109=1231.738,8.962,-41.510,-179.346,5.315,148.725
C05110=1231.743,8.713,-41.495,-179.348,5.315,148.725
C05111=1231.748,8.463,-41.481,-179.350,5.314,148.726
C05112=1231.752,8.214,-41.466,-179.353,5.314,148.727
C05113=1231.758,7.964,-41.451,-179.356,5.313,148.727
C05114=1231.763,7.715,-41.436,-179.358,5.314,148.728
C05115=1231.768,7.465,-41.421,-179.360,5.313,148.729
C05116=1231.773,7.216,-41.406,-179.363,5.313,148.729
C05117=1231.778,6.966,-41.392,-179.366,5.312,148.730
C05118=1231.783,6.717,-41.377,-179.368,5.312,148.731
C05119=1231.788,6.467,-41.362,-179.370,5.312,148.731
C05120=1231.793,6.218,-41.347,-179.373,5.311,148.732
C05121=1231.798,5.968,-41.332,-179.375,5.311,148.733
C05122=1231.803,5.718,-41.318,-179.378,5.311,148.733
C05123=1231.808,5.469,-41.303,-179.380,5.310,148.734
C05124=1231.813,5.219,-41.288,-179.383,5.310,148.735
C05125=1231.818,4.970,-41.273,-179.385,5.310,148.736
C05126=1231.823,4.721,-41.259,-179.388,5.310,148.736
C05127=1231.828,4.471,-41.244,-179.391,5.309,148.737
C05128=1231.833,4.221,-41.229,-179.393,5.309,148.738
C05129=1231.838,3.953,-41.213,-179.395,5.309,148.738
C05130=1231.844,3.684,-41.198,-179.398,5.308,148.739
C05131=1231.849,3.415,-41.181,-179.401,5.308,148.740
C05132=1231.855,3.146,-41.166,-179.404,5.308,148.741
C05133=1231.859,2.896,-41.151,-179.406,5.307,148.741
C05134=1231.864,2.647,-41.137,-179.408,5.307,148.742
C05135=1231.869,2.397,-41.122,-179.411,5.307,148.743
C05136=1231.875,2.147,-41.107,-179.414,5.306,148.743
C05137=1231.880,1.898,-41.093,-179.416,5.306,148.744
C05138=1231.884,1.649,-41.078,-179.418,5.306,148.745
C05139=1231.889,1.399,-41.064,-179.421,5.306,148.745
C05140=1231.894,1.149,-41.049,-179.424,5.305,148.746
C05141=1231.899,0.900,-41.035,-179.426,5.305,148.747
C05142=1231.904,0.651,-41.021,-179.429,5.305,148.747
C05143=1231.910,0.401,-41.006,-179.431,5.304,148.748
C05144=1231.915,0.151,-40.991,-179.434,5.304,148.749
C05145=1231.920,-0.098,-40.976,-179.436,5.304,148.750
C05146=1231.925,-0.347,-40.962,-179.439,5.303,148.750
C05147=1231.930,-0.597,-40.948,-179.441,5.303,148.751
C05148=1231.935,-0.847,-40.934,-179.443,5.303,148.752
C05149=1231.940,-1.097,-40.919,-179.446,5.303,148.752
C05150=1231.944,-1.346,-40.904,-179.449,5.302,148.753
C05151=1231.950,-1.596,-40.889,-179.451,5.302,148.754
C05152=1231.955,-1.845,-40.876,-179.453,5.302,148.754
C05153=1231.960,-2.094,-40.861,-179.456,5.301,148.755
C05154=1231.965,-2.344,-40.847,-179.459,5.301,148.756
C05155=1231.970,-2.593,-40.832,-179.461,5.301,148.756
C05156=1231.975,-2.843,-40.818,-179.463,5.301,148.757
C05157=1231.980,-3.093,-40.803,-179.466,5.300,148.758
C05158=1231.985,-3.342,-40.789,-179.468,5.300,148.758
C05159=1231.990,-3.592,-40.775,-179.471,5.300,148.759
C05160=1231.995,-3.841,-40.761,-179.473,5.299,148.760
C05161=1232.000,-4.090,-40.746,-179.476,5.299,148.761
C05162=1232.005,-4.340,-40.732,-179.478,5.299,148.761
C05163=1232.010,-4.590,-40.717,-179.481,5.299,148.762
C05164=1232.015,-4.839,-40.703,-179.484,5.298,148.763
C05165=1232.020,-5.089,-40.689,-179.486,5.299,148.764
C05166=1232.025,-5.338,-40.675,-179.489,5.298,148.764
C05167=1232.030,-5.588,-40.661,-179.491,5.298,148.765
C05168=1232.035,-5.837,-40.646,-179.493,5.298,148.766
C05169=1232.040,-6.087,-40.632,-179.496,5.297,148.766
C05170=1232.045,-6.337,-40.618,-179.499,5.297,148.767
C05171=1232.050,-6.586,-40.603,-179.501,5.297,148.768
C05172=1232.055,-6.835,-40.589,-179.503,5.297,148.768
C05173=1232.060,-7.085,-40.575,-179.506,5.296,148.769
C05174=1232.065,-7.334,-40.560,-179.509,5.296,148.770
C05175=1232.070,-7.584,-40.546,-179.511,5.296,148.770
C05176=1232.075,-7.834,-40.532,-179.513,5.295,148.771
C05177=1232.081,-8.083,-40.518,-179.516,5.295,148.772
C05178=1232.086,-8.332,-40.504,-179.518,5.295,148.773
C05179=1232.091,-8.582,-40.489,-179.521,5.295,148.773
C05180=1232.096,-8.832,-40.475,-179.524,5.294,148.774
C05181=1232.101,-9.082,-40.461,-179.526,5.294,148.775
C05182=1232.106,-9.331,-40.447,-179.528,5.294,148.775
C05183=1232.111,-9.580,-40.433,-179.531,5.293,148.776
C05184=1232.116,-9.830,-40.418,-179.533,5.294,148.777
C05185=1232.120,-10.079,-40.405,-179.536,5.293,148.777
C05186=1232.126,-10.329,-40.391,-179.538,5.293,148.778
C05187=1232.131,-10.579,-40.377,-179.540,5.293,148.779
C05188=1232.136,-10.828,-40.363,-179.543,5.292,148.779
C05189=1232.141,-11.078,-40.349,-179.546,5.292,148.780
C05190=1232.147,-11.327,-40.335,-179.548,5.292,148.781
C05191=1232.152,-11.577,-40.320,-179.550,5.292,148.782
C05192=1232.157,-11.827,-40.306,-179.553,5.291,148.782
C05193=1232.161,-12.076,-40.292,-179.555,5.291,148.783
C05194=1232.166,-12.325,-40.279,-179.558,5.291,148.784
C05195=1232.171,-12.575,-40.264,-179.561,5.291,148.785
C05196=1232.176,-12.824,-40.250,-179.563,5.291,148.785
C05197=1232.181,-13.075,-40.236,-179.566,5.290,148.786
C05198=1232.187,-13.324,-40.223,-179.568,5.290,148.787
C05199=1232.192,-13.574,-40.208,-179.570,5.290,148.787
C05200=1232.196,-13.823,-40.195,-179.573,5.290,148.788
C05201=1232.201,-14.073,-40.180,-179.576,5.289,148.789
C05202=1232.207,-14.322,-40.166,-179.578,5.290,148.789
C05203=1232.212,-14.572,-40.153,-179.581,5.289,148.790
C05204=1232.217,-14.822,-40.139,-179.583,5.288,148.791
C05205=1232.222,-15.071,-40.125,-179.585,5.289,148.791
C05206=1232.227,-15.320,-40.111,-179.588,5.288,148.792
C05207=1232.232,-15.570,-40.097,-179.591,5.288,148.793
C05208=1232.238,-15.819,-40.083,-179.593,5.288,148.794
C05209=1232.242,-16.069,-40.069,-179.595,5.288,148.794
C05210=1232.247,-16.319,-40.055,-179.598,5.287,148.795
C05211=1232.252,-16.568,-40.042,-179.600,5.287,148.796
C05212=1232.258,-16.818,-40.028,-179.603,5.287,148.796
C05213=1232.262,-17.068,-40.014,-179.605,5.286,148.797
C05214=1232.268,-17.317,-40.000,-179.607,5.287,148.798
C05215=1232.272,-17.566,-39.986,-179.610,5.286,148.798
C05216=1232.278,-17.816,-39.973,-179.613,5.286,148.799
C05217=1232.283,-18.065,-39.959,-179.615,5.286,148.800
C05218=1232.288,-18.315,-39.944,-179.618,5.286,148.801
C05219=1232.293,-18.565,-39.931,-179.621,5.285,148.801
C05220=1232.298,-18.814,-39.918,-179.623,5.285,148.802
C05221=1232.303,-19.064,-39.903,-179.625,5.285,148.803
C05222=1232.308,-19.314,-39.890,-179.627,5.285,148.804
C05223=1232.313,-19.563,-39.876,-179.630,5.285,148.804
C05224=1232.318,-19.813,-39.862,-179.633,5.284,148.805
C05225=1232.323,-20.063,-39.849,-179.635,5.285,148.806
C05226=1232.328,-20.312,-39.835,-179.638,5.284,148.806
C05227=1232.333,-20.561,-39.821,-179.640,5.284,148.807
C05228=1232.339,-20.811,-39.808,-179.642,5.284,148.808
C05229=1232.343,-21.060,-39.794,-179.645,5.283,148.808
C05230=1232.348,-21.310,-39.780,-179.648,5.283,148.809
C05231=1232.354,-21.560,-39.767,-179.650,5.283,148.810
C05232=1232.358,-21.809,-39.753,-179.652,5.283,148.810
C05233=1232.364,-22.078,-39.738,-179.655,5.282,148.811
C05234=1232.370,-22.348,-39.724,-179.658,5.283,148.812
C05235=1232.375,-22.617,-39.709,-179.660,5.282,148.813
C05236=1232.381,-22.887,-39.694,-179.663,5.282,148.813
C05237=1232.386,-23.135,-39.681,-179.666,5.281,148.814
C05238=1232.391,-23.386,-39.667,-179.668,5.282,148.815
C05239=1232.395,-23.635,-39.653,-179.670,5.281,148.816
C05240=1232.401,-23.885,-39.640,-179.673,5.281,148.816
C05241=1232.406,-24.134,-39.626,-179.676,5.281,148.817
C05242=1232.411,-24.384,-39.613,-179.678,5.281,148.818
C05243=1232.416,-24.633,-39.599,-179.680,5.281,148.819
C05244=1232.421,-24.883,-39.587,-179.683,5.280,148.819
C05245=1232.426,-25.132,-39.572,-179.686,5.280,148.820
C05246=1232.431,-25.383,-39.559,-179.688,5.280,148.821
C05247=1232.436,-25.631,-39.545,-179.690,5.280,148.821
C05248=1232.441,-25.882,-39.532,-179.693,5.279,148.822
C05249=1232.446,-26.130,-39.518,-179.695,5.280,148.823
C05250=1232.452,-26.381,-39.505,-179.698,5.279,148.823
C05251=1232.456,-26.629,-39.492,-179.700,5.279,148.824
C05252=1232.462,-26.880,-39.478,-179.702,5.279,148.825
C05253=1232.466,-27.129,-39.465,-179.705,5.278,148.826
C05254=1232.472,-27.379,-39.451,-179.707,5.279,148.826
C05255=1232.477,-27.628,-39.437,-179.710,5.278,148.827
C05256=1232.482,-27.878,-39.424,-179.713,5.278,148.828
C05257=1232.488,-28.128,-39.411,-179.715,5.278,148.828
C05258=1232.492,-28.377,-39.397,-179.717,5.277,148.829
C05259=1232.498,-28.627,-39.384,-179.719,5.278,148.830
C05260=1232.502,-28.876,-39.371,-179.722,5.277,148.830
C05261=1232.508,-29.126,-39.357,-179.725,5.277,148.831
C05262=1232.512,-29.376,-39.344,-179.727,5.277,148.832
C05263=1232.518,-29.625,-39.330,-179.730,5.277,148.833
C05264=1232.522,-29.875,-39.317,-179.733,5.276,148.833
C05265=1232.528,-30.124,-39.304,-179.735,5.277,148.834
C05266=1232.532,-30.374,-39.291,-179.737,5.276,148.835
C05267=1232.538,-30.623,-39.277,-179.739,5.277,148.836
C05268=1232.543,-30.873,-39.264,-179.742,5.276,148.836
C05269=1232.548,-31.122,-39.251,-179.745,5.276,148.837
C05270=1232.553,-31.372,-39.238,-179.747,5.276,148.838
C05271=1232.558,-31.622,-39.225,-179.749,5.275,148.838
C05272=1232.563,-31.871,-39.211,-179.752,5.276,148.839
C05273=1232.568,-32.121,-39.198,-179.754,5.275,148.840
C05274=1232.573,-32.371,-39.185,-179.757,5.275,148.840
C05275=1232.579,-32.620,-39.172,-179.759,5.275,148.841
C05276=1232.583,-32.870,-39.158,-179.762,5.274,148.842
C05277=1232.589,-33.119,-39.145,-179.764,5.275,148.843
C05278=1232.594,-33.369,-39.132,-179.766,5.274,148.843
C05279=1232.599,-33.619,-39.119,-179.769,5.274,148.844
C05280=1232.604,-33.868,-39.106,-179.771,5.274,148.845
C05281=1232.609,-34.118,-39.092,-179.774,5.274,148.845
C05282=1232.614,-34.367,-39.079,-179.777,5.273,148.846
C05283=1232.619,-34.617,-39.066,-179.779,5.274,148.847
C05284=1232.624,-34.866,-39.053,-179.782,5.273,148.848
C05285=1232.629,-35.116,-39.040,-179.784,5.274,148.848
C05286=1232.635,-35.366,-39.026,-179.786,5.273,148.849
C05287=1232.640,-35.615,-39.014,-179.789,5.273,148.850
C05288=1232.644,-35.865,-39.001,-179.791,5.273,148.850
C05289=1232.650,-36.114,-38.987,-179.794,5.272,148.851
C05290=1232.655,-36.364,-38.974,-179.796,5.273,148.852
C05291=1232.660,-36.614,-38.961,-179.799,5.272,148.853
C05292=1232.665,-36.863,-38.948,-179.801,5.272,148.853
C05293=1232.670,-37.113,-38.935,-179.803,5.272,148.854
C05294=1232.675,-37.363,-38.923,-179.806,5.271,148.855
C05295=1232.681,-37.612,-38.909,-179.808,5.272,148.855
C05296=1232.685,-37.862,-38.896,-179.811,5.271,148.856
C05297=1232.690,-38.111,-38.883,-179.813,5.272,148.857
C05298=1232.696,-38.361,-38.870,-179.815,5.271,148.857
C05299=1232.701,-38.611,-38.857,-179.818,5.271,148.858
C05300=1232.706,-38.860,-38.844,-179.820,5.271,148.859
C05301=1232.711,-39.110,-38.831,-179.823,5.271,148.860
C05302=1232.716,-39.360,-38.818,-179.825,5.271,148.860
C05303=1232.721,-39.609,-38.806,-179.828,5.271,148.861
C05304=1232.726,-39.859,-38.793,-179.831,5.270,148.862
C05305=1232.732,-40.109,-38.779,-179.833,5.270,148.863
C05306=1232.737,-40.358,-38.767,-179.836,5.270,148.863
C05307=1232.741,-40.608,-38.754,-179.838,5.270,148.864
C05308=1232.747,-40.858,-38.741,-179.840,5.270,148.865
C05309=1232.752,-41.107,-38.728,-179.843,5.269,148.865
C05310=1232.757,-41.357,-38.715,-179.845,5.270,148.866
C05311=1232.762,-41.606,-38.702,-179.848,5.269,148.867
C05312=1232.768,-41.856,-38.689,-179.850,5.269,148.867
C05313=1232.772,-42.106,-38.676,-179.852,5.269,148.868
C05314=1232.777,-42.355,-38.664,-179.855,5.269,148.869
C05315=1232.783,-42.604,-38.651,-179.857,5.269,148.870
C05316=1232.787,-42.855,-38.638,-179.860,5.268,148.870
C05317=1232.793,-43.104,-38.625,-179.862,5.269,148.871
C05318=1232.798,-43.353,-38.612,-179.865,5.268,148.872
C05319=1232.803,-43.603,-38.599,-179.867,5.268,148.872
C05320=1232.808,-43.853,-38.587,-179.869,5.268,148.873
C05321=1232.813,-44.102,-38.574,-179.873,5.268,148.874
C05322=1232.819,-44.352,-38.561,-179.875,5.268,148.875
C05323=1232.823,-44.602,-38.548,-179.877,5.268,148.875
C05324=1232.828,-44.851,-38.535,-179.879,5.268,148.876
C05325=1232.833,-45.100,-38.523,-179.882,5.267,148.877
C05326=1232.838,-45.350,-38.510,-179.884,5.268,148.878
C05327=1232.843,-45.600,-38.497,-179.887,5.267,148.878
C05328=1232.849,-45.849,-38.484,-179.889,5.267,148.879
C05329=1232.854,-46.099,-38.472,-179.892,5.267,148.880
C05330=1232.859,-46.349,-38.459,-179.894,5.267,148.880
C05331=1232.864,-46.599,-38.447,-179.896,5.267,148.881
C05332=1232.869,-46.848,-38.434,-179.899,5.266,148.882
C05333=1232.874,-47.097,-38.421,-179.901,5.267,148.882
C05334=1232.879,-47.347,-38.408,-179.904,5.266,148.883
C05335=1232.885,-47.597,-38.395,-179.906,5.266,148.884
C05336=1232.890,-47.847,-38.383,-179.908,5.266,148.885
C05337=1232.895,-48.117,-38.370,-179.912,5.266,148.886
C05338=1232.901,-48.386,-38.356,-179.914,5.266,148.886
C05339=1232.906,-48.656,-38.342,-179.916,5.266,148.887
C05340=1232.911,-48.925,-38.328,-179.919,5.265,148.888
C05341=1232.917,-49.175,-38.317,-179.922,5.266,148.889
C05342=1232.922,-49.425,-38.304,-179.924,5.266,148.889
C05343=1232.927,-49.674,-38.291,-179.927,5.265,148.890
C05344=1232.932,-49.924,-38.278,-179.929,5.265,148.891
C05345=1232.938,-50.174,-38.266,-179.932,5.265,148.891
C05346=1232.943,-50.424,-38.253,-179.934,5.265,148.892
C05347=1232.948,-50.673,-38.241,-179.936,5.265,148.893
C05348=1232.953,-50.922,-38.228,-179.939,5.265,148.893
C05349=1232.958,-51.173,-38.216,-179.941,5.265,148.894
C05350=1232.963,-51.422,-38.203,-179.944,5.264,148.895
C05351=1232.968,-51.671,-38.191,-179.946,5.264,148.896
C05352=1232.973,-51.921,-38.178,-179.949,5.264,148.896
C05353=1232.979,-52.171,-38.166,-179.951,5.264,148.897
C05354=1232.983,-52.421,-38.153,-179.953,5.264,148.898
C05355=1232.988,-52.670,-38.141,-179.955,5.264,148.898
C05356=1232.994,-52.920,-38.129,-179.958,5.264,148.899
C05357=1232.999,-53.169,-38.116,-179.960,5.264,148.900
C05358=1233.004,-53.419,-38.103,-179.963,5.263,148.901
C05359=1233.010,-53.669,-38.092,-179.966,5.263,148.901
C05360=1233.014,-53.919,-38.079,-179.968,5.263,148.902
C05361=1233.019,-54.168,-38.066,-179.970,5.263,148.903
C05362=1233.025,-54.418,-38.054,-179.973,5.264,148.904
C05363=1233.030,-54.667,-38.042,-179.976,5.263,148.904
C05364=1233.035,-54.916,-38.029,-179.978,5.263,148.905
C05365=1233.040,-55.166,-38.017,-179.980,5.263,148.906
C05366=1233.045,-55.416,-38.004,-179.982,5.263,148.906
C05367=1233.050,-55.666,-37.992,-179.985,5.263,148.907
C05368=1233.055,-55.915,-37.980,-179.988,5.262,148.908
C05369=1233.060,-56.165,-37.968,-179.990,5.263,148.908
C05370=1233.065,-56.415,-37.956,-179.992,5.262,148.909
C05371=1233.070,-56.664,-37.943,-179.995,5.262,148.910
C05372=1233.076,-56.914,-37.931,-179.997,5.262,148.911
C05373=1233.080,-57.164,-37.918,-179.999,5.262,148.911
C05374=1233.085,-57.413,-37.906,179.998,5.262,148.912
C05375=1233.091,-57.663,-37.894,179.996,5.262,148.913
C05376=1233.096,-57.912,-37.881,179.993,5.262,148.913
C05377=1233.101,-58.162,-37.869,179.991,5.262,148.914
C05378=1233.107,-58.412,-37.857,179.988,5.261,148.915
C05379=1233.111,-58.661,-37.845,179.986,5.261,148.916
C05380=1233.116,-58.911,-37.833,179.984,5.261,148.916
C05381=1233.122,-59.161,-37.821,179.981,5.261,148.917
C05382=1233.127,-59.410,-37.808,179.979,5.261,148.918
C05383=1233.132,-59.661,-37.796,179.976,5.261,148.918
C05384=1233.137,-59.910,-37.783,179.974,5.261,148.919
C05385=1233.142,-60.160,-37.772,179.971,5.261,148.920
C05386=1233.147,-60.409,-37.759,179.969,5.261,148.921
C05387=1233.152,-60.659,-37.748,179.966,5.261,148.921
C05388=1233.157,-60.908,-37.735,179.964,5.261,148.922
C05389=1233.163,-61.158,-37.723,179.962,5.261,148.923
C05390=1233.168,-61.408,-37.711,179.959,5.261,148.924
C05391=1233.173,-61.657,-37.699,179.957,5.260,148.924
C05392=1233.179,-61.907,-37.687,179.954,5.260,148.925
C05393=1233.183,-62.156,-37.675,179.952,5.260,148.926
C05394=1233.188,-62.406,-37.663,179.949,5.260,148.926
C05395=1233.194,-62.655,-37.650,179.947,5.260,148.927
C05396=1233.199,-62.905,-37.638,179.945,5.260,148.928
C05397=1233.204,-63.155,-37.627,179.943,5.260,148.928
C05398=1233.209,-63.404,-37.615,179.940,5.260,148.929
C05399=1233.214,-63.654,-37.603,179.938,5.260,148.930
C05400=1233.219,-63.904,-37.590,179.935,5.259,148.931
C05401=1233.225,-64.153,-37.578,179.933,5.260,148.931
C05402=1233.229,-64.403,-37.567,179.930,5.259,148.932
C05403=1233.235,-64.652,-37.554,179.928,5.260,148.933
C05404=1233.240,-64.902,-37.542,179.926,5.259,148.933
C05405=1233.245,-65.152,-37.531,179.923,5.259,148.934
C05406=1233.251,-65.402,-37.518,179.921,5.259,148.935
C05407=1233.255,-65.651,-37.507,179.918,5.259,148.936
C05408=1233.261,-65.901,-37.495,179.916,5.259,148.936
C05409=1233.266,-66.151,-37.482,179.913,5.258,148.937
C05410=1233.271,-66.400,-37.470,179.911,5.259,148.938
C05411=1233.276,-66.650,-37.459,179.909,5.258,148.938
C05412=1233.281,-66.900,-37.447,179.906,5.259,148.939
C05413=1233.286,-67.149,-37.434,179.903,5.258,148.940
C05414=1233.291,-67.399,-37.423,179.901,5.259,148.941
C05415=1233.297,-67.649,-37.411,179.899,5.258,148.941
C05416=1233.302,-67.899,-37.399,179.897,5.259,148.942
C05417=1233.307,-68.148,-37.387,179.894,5.258,148.943
C05418=1233.312,-68.398,-37.376,179.892,5.259,148.944
C05419=1233.317,-68.648,-37.364,179.889,5.258,148.944
C05420=1233.323,-68.898,-37.352,179.887,5.258,148.945
C05421=1233.327,-69.147,-37.340,179.884,5.258,148.946
C05422=1233.333,-69.397,-37.328,179.882,5.258,148.946
C05423=1233.338,-69.647,-37.316,179.880,5.258,148.947
C05424=1233.343,-69.896,-37.305,179.878,5.258,148.948
C05425=1233.348,-70.146,-37.293,179.875,5.258,148.948
C05426=1233.353,-70.395,-37.280,179.873,5.258,148.949
C05427=1233.358,-70.645,-37.269,179.870,5.258,148.950
C05428=1233.363,-70.895,-37.257,179.868,5.258,148.951
C05429=1233.369,-71.145,-37.245,179.865,5.257,148.951
C05430=1233.373,-71.395,-37.234,179.863,5.257,148.952
C05431=1233.379,-71.644,-37.222,179.861,5.257,148.953
C05432=1233.384,-71.893,-37.210,179.858,5.257,148.953
C05433=1233.389,-72.143,-37.198,179.856,5.257,148.954
C05434=1233.395,-72.393,-37.187,179.853,5.257,148.955
C05435=1233.399,-72.642,-37.175,179.851,5.257,148.956
C05436=1233.405,-72.892,-37.163,179.848,5.257,148.956
C05437=1233.410,-73.142,-37.151,179.846,5.257,148.957
C05438=1233.415,-73.392,-37.140,179.844,5.256,148.958
C05439=1233.420,-73.642,-37.128,179.842,5.257,148.958
C05440=1233.425,-73.891,-37.116,179.839,5.256,148.959
C05441=1233.431,-74.161,-37.104,179.836,5.257,148.960
C05442=1233.436,-74.431,-37.091,179.834,5.257,148.961
C05443=1233.442,-74.701,-37.079,179.831,5.256,148.961
C05444=1233.448,-74.972,-37.067,179.829,5.256,148.962
C05445=1233.453,-75.222,-37.055,179.826,5.256,148.963
C05446=1233.458,-75.472,-37.043,179.824,5.256,148.964
C05447=1233.463,-75.721,-37.032,179.821,5.256,148.964
C05448=1233.468,-75.971,-37.020,179.819,5.256,148.965
C05449=1233.474,-76.220,-37.009,179.816,5.256,148.966
C05450=1233.479,-76.470,-36.997,179.814,5.256,148.967
C05451=1233.484,-76.720,-36.986,179.811,5.256,148.967
C05452=1233.490,-76.970,-36.974,179.809,5.256,148.968
C05453=1233.494,-77.219,-36.962,179.807,5.256,148.969
C05454=1233.500,-77.469,-36.951,179.805,5.256,148.969
C05455=1233.505,-77.718,-36.940,179.802,5.256,148.970
C05456=1233.511,-77.968,-36.928,179.800,5.256,148.971
C05457=1233.515,-78.218,-36.916,179.797,5.256,148.972
C05458=1233.521,-78.468,-36.905,179.795,5.256,148.972
C05459=1233.525,-78.717,-36.893,179.792,5.255,148.973
C05460=1233.531,-78.967,-36.881,179.790,5.256,148.974
C05461=1233.536,-79.216,-36.870,179.788,5.255,148.974
C05462=1233.541,-79.466,-36.859,179.785,5.256,148.975
C05463=1233.546,-79.716,-36.847,179.783,5.255,148.976
C05464=1233.551,-79.965,-36.836,179.781,5.256,148.977
C05465=1233.556,-80.215,-36.824,179.778,5.255,148.977
C05466=1233.562,-80.464,-36.813,179.776,5.255,148.978
C05467=1233.567,-80.714,-36.801,179.773,5.255,148.979
C05468=1233.572,-80.964,-36.790,179.771,5.255,148.979
C05469=1233.577,-81.214,-36.779,179.768,5.255,148.980
C05470=1233.582,-81.464,-36.768,179.766,5.255,148.981
C05471=1233.587,-81.713,-36.757,179.764,5.255,148.982
C05472=1233.593,-81.963,-36.745,179.762,5.255,148.982
C05473=1233.598,-82.213,-36.733,179.759,5.255,148.983
C05474=1233.603,-82.463,-36.722,179.757,5.255,148.984
C05475=1233.608,-82.712,-36.710,179.754,5.255,148.984
C05476=1233.613,-82.962,-36.700,179.752,5.255,148.985
C05477=1233.619,-83.212,-36.688,179.749,5.254,148.986
C05478=1233.623,-83.461,-36.677,179.747,5.255,148.987
